LIN {X 0,Y 411.191,Z 465.266,A -85,B 0,C 180,E1 -10409.152,E2 -10409.152} C_VEL
LIN {X 0,Y 411.26,Z 465.255,A -85,B 0,C 180,E1 -10412.522,E2 -10412.522} C_VEL
LIN {X 0,Y 411.229,Z 465.262,A -85,B 0,C 180,E1 -10415.784,E2 -10415.784} C_VEL
LIN {X 0,Y 411.198,Z 465.264,A -85,B 0,C 180,E1 -10418.966,E2 -10418.966} C_VEL
LIN {X 0,Y 411.254,Z 465.257,A -85,B 0,C 180,E1 -10422.085,E2 -10422.085} C_VEL
LIN {X 0,Y 411.262,Z 465.258,A -85,B 0,C 180,E1 -10425.147,E2 -10425.147} C_VEL
LIN {X 0,Y 411.285,Z 465.252,A -85,B 0,C 180,E1 -10428.167,E2 -10428.167} C_VEL
LIN {X 0,Y 411.483,Z 465.229,A -85,B 0,C 180,E1 -10432.146,E2 -10432.146} C_VEL
LIN {X 0,Y 411.476,Z 465.229,A -85,B 0,C 180,E1 -10434.118,E2 -10434.118} C_VEL
LIN {X 0,Y 411.515,Z 465.226,A -85,B 0,C 180,E1 -10438.042,E2 -10438.042} C_VEL
LIN {X 0,Y 411.643,Z 465.21,A -85,B 0,C 180,E1 -10440,E2 -10440} C_VEL
LIN {X 0,Y 411.459,Z 465.231,A -85,B 0,C 180,E1 -10442.937,E2 -10442.937} C_VEL
LIN {X 0,Y 411.461,Z 465.232,A -85,B 0,C 180,E1 -10446.867,E2 -10446.867} C_VEL
LIN {X 0,Y 411.293,Z 465.252,A -85,B 0,C 180,E1 -10449.839,E2 -10449.839} C_VEL
LIN {X 0,Y 411.306,Z 465.253,A -85,B 0,C 180,E1 -10453.104,E2 -10453.104} C_VEL
LIN {X 0,Y 411.263,Z 465.255,A -85,B 0,C 180,E1 -10456.869,E2 -10456.869} C_VEL
LIN {X 0,Y 411.231,Z 465.261,A -85,B 0,C 180,E1 -10459.987,E2 -10459.987} C_VEL
LIN {X 0,Y 411.204,Z 465.264,A -85,B 0,C 180,E1 -10463.147,E2 -10463.147} C_VEL
LIN {X 0,Y 411.238,Z 465.258,A -85,B 0,C 180,E1 -10466.381,E2 -10466.381} C_VEL
LIN {X 0,Y 411.2,Z 465.266,A -85,B 0,C 180,E1 -10469.713,E2 -10469.713} C_VEL
LIN {X 0,Y 411.206,Z 465.266,A -85,B 0,C 180,E1 -10473.156,E2 -10473.156} C_VEL
LIN {X 0,Y 411.195,Z 465.264,A -85,B 0,C 180,E1 -10476.553,E2 -10476.553} C_VEL
LIN {X 0,Y 411.217,Z 465.262,A -85,B 0,C 180,E1 -10479.729,E2 -10479.729} C_VEL
LIN {X 0,Y 411.231,Z 465.262,A -85,B 0,C 180,E1 -10483.126,E2 -10483.126} C_VEL
LIN {X 0,Y 411.172,Z 465.275,A -85,B 0,C 180,E1 -10485.881,E2 -10485.881} C_VEL
LIN {X 0,Y 411.284,Z 465.464,A -85,B 0,C 180,E1 -10487.44,E2 -10487.44} C_VEL
LIN {X 0,Y 412.469,Z 472.197,A -85,B 0,C 180,E1 -10490.918,E2 -10490.918} C_VEL
LIN {X 0,Y 413.284,Z 477.387,A -85,B 0,C 180,E1 -10493.474,E2 -10493.474} C_VEL
LIN {X 0,Y 413.079,Z 482.509,A -85,B 0,C 180,E1 -10495.844,E2 -10495.844} C_VEL
LIN {X 0,Y 412.407,Z 490.177,A -85,B 0,C 180,E1 -10499.254,E2 -10499.254} C_VEL
LIN {X 0,Y 411.822,Z 497.821,A -85,B 0,C 180,E1 -10502.563,E2 -10502.563} C_VEL
LIN {X 0,Y 411.283,Z 505.453,A -85,B 0,C 180,E1 -10505.788,E2 -10505.788} C_VEL
LIN {X 0,Y 410.808,Z 514.359,A -85,B 0,C 180,E1 -10509.47,E2 -10509.47} C_VEL
LIN {X 0,Y 410.523,Z 522.363,A -85,B 0,C 180,E1 -10512.726,E2 -10512.726} C_VEL
LIN {X 0,Y 412.529,Z 536.719,A -85,B 0,C 180,E1 -10513.296,E2 -10513.296} C_VEL
LIN {X 0,Y 413.816,Z 548.267,A -85,B 0,C 180,E1 -10513.913,E2 -10513.913} C_VEL
LIN {X 0,Y 414.068,Z 553.582,A -85,B 0,C 180,E1 -10514.243,E2 -10514.243} C_VEL
LIN {X 0,Y 413.319,Z 565.526,A -85,B 0,C 180,E1 -10515.097,E2 -10515.097} C_VEL
LIN {X 0,Y 412.57,Z 576.424,A -85,B 0,C 180,E1 -10516.077,E2 -10516.077} C_VEL
LIN {X 0,Y 411.928,Z 586.371,A -85,B 0,C 180,E1 -10517.186,E2 -10517.186} C_VEL
LIN {X 0,Y 411.336,Z 595.435,A -85,B 0,C 180,E1 -10518.419,E2 -10518.419} C_VEL
LIN {X 0,Y 410.758,Z 604.315,A -85,B 0,C 180,E1 -10519.9,E2 -10519.9} C_VEL
LIN {X 0,Y 410.401,Z 611.44,A -85,B 0,C 180,E1 -10521.382,E2 -10521.382} C_VEL
LIN {X 0,Y 410.162,Z 617.937,A -85,B 0,C 180,E1 -10523.111,E2 -10523.111} C_VEL
LIN {X 0,Y 410.08,Z 622.193,A -85,B 0,C 180,E1 -10524.591,E2 -10524.591} C_VEL
LIN {X 0,Y 409.976,Z 625.337,A -85,B 0,C 180,E1 -10526.068,E2 -10526.068} C_VEL
LIN {X 0,Y 410.07,Z 626.893,A -85,B 0,C 180,E1 -10527.053,E2 -10527.053} C_VEL
LIN {X 0,Y 410.058,Z 627.975,A -85,B 0,C 180,E1 -10528.036,E2 -10528.036} C_VEL
LIN {X 0,Y 410.037,Z 628.624,A -85,B 0,C 180,E1 -10529.018,E2 -10529.018} C_VEL
LIN {X 0,Y 410.047,Z 628.868,A -85,B 0,C 180,E1 -10530,E2 -10530} C_VEL
LIN {X 0,Y 410.026,Z 628.7,A -85,B 0,C 180,E1 -10530.982,E2 -10530.982} C_VEL
LIN {X 0,Y 410.059,Z 628.077,A -85,B 0,C 180,E1 -10531.965,E2 -10531.965} C_VEL
LIN {X 0,Y 410.045,Z 627.032,A -85,B 0,C 180,E1 -10532.948,E2 -10532.948} C_VEL
LIN {X 0,Y 409.979,Z 625.569,A -85,B 0,C 180,E1 -10533.932,E2 -10533.932} C_VEL
LIN {X 0,Y 410.043,Z 622.528,A -85,B 0,C 180,E1 -10535.409,E2 -10535.409} C_VEL
LIN {X 0,Y 410.164,Z 618.421,A -85,B 0,C 180,E1 -10536.889,E2 -10536.889} C_VEL
LIN {X 0,Y 410.444,Z 612.154,A -85,B 0,C 180,E1 -10538.617,E2 -10538.617} C_VEL
LIN {X 0,Y 410.83,Z 604.043,A -85,B 0,C 180,E1 -10540.348,E2 -10540.348} C_VEL
LIN {X 0,Y 411.507,Z 595.34,A -85,B 0,C 180,E1 -10541.826,E2 -10541.826} C_VEL
LIN {X 0,Y 412.242,Z 584.879,A -85,B 0,C 180,E1 -10543.262,E2 -10543.262} C_VEL
LIN {X 0,Y 413.051,Z 574.993,A -85,B 0,C 180,E1 -10544.372,E2 -10544.372} C_VEL
LIN {X 0,Y 413.928,Z 563.907,A -85,B 0,C 180,E1 -10545.385,E2 -10545.385} C_VEL
LIN {X 0,Y 414.759,Z 552.383,A -85,B 0,C 180,E1 -10546.236,E2 -10546.236} C_VEL
LIN {X 0,Y 413.894,Z 539.48,A -85,B 0,C 180,E1 -10547.068,E2 -10547.068} C_VEL
LIN {X 0,Y 412.163,Z 526.898,A -85,B 0,C 180,E1 -10547.744,E2 -10547.744} C_VEL
LIN {X 0,Y 410.508,Z 518.922,A -85,B 0,C 180,E1 -10548.142,E2 -10548.142} C_VEL
LIN {X 0,Y 410.885,Z 510.509,A -85,B 0,C 180,E1 -10551.577,E2 -10551.577} C_VEL
LIN {X 0,Y 411.362,Z 501.923,A -85,B 0,C 180,E1 -10555.285,E2 -10555.285} C_VEL
LIN {X 0,Y 411.912,Z 494.917,A -85,B 0,C 180,E1 -10558.538,E2 -10558.538} C_VEL
LIN {X 0,Y 412.708,Z 488.374,A -85,B 0,C 180,E1 -10561.864,E2 -10561.864} C_VEL
LIN {X 0,Y 413.241,Z 484.363,A -85,B 0,C 180,E1 -10564.141,E2 -10564.141} C_VEL
LIN {X 0,Y 413.602,Z 480.707,A -85,B 0,C 180,E1 -10566.493,E2 -10566.493} C_VEL
LIN {X 0,Y 413.341,Z 477.537,A -85,B 0,C 180,E1 -10568.985,E2 -10568.985} C_VEL
LIN {X 0,Y 412.897,Z 474.939,A -85,B 0,C 180,E1 -10571.593,E2 -10571.593} C_VEL
LIN {X 0,Y 412.566,Z 472.95,A -85,B 0,C 180,E1 -10574.319,E2 -10574.319} C_VEL
LIN {X 0,Y 412.337,Z 471.651,A -85,B 0,C 180,E1 -10577.131,E2 -10577.131} C_VEL
LIN {X 0,Y 412.148,Z 471.064,A -85,B 0,C 180,E1 -10580.117,E2 -10580.117} C_VEL
LIN {X 0,Y 412.09,Z 471.198,A -85,B 0,C 180,E1 -10583.351,E2 -10583.351} C_VEL
LIN {X 0,Y 411.907,Z 471.748,A -85,B 0,C 180,E1 -10585.733,E2 -10585.733} C_VEL
LIN {X 0,Y 411.595,Z 473.076,A -85,B 0,C 180,E1 -10589.186,E2 -10589.186} C_VEL
LIN {X 0,Y 411.225,Z 474.94,A -85,B 0,C 180,E1 -10592.711,E2 -10592.711} C_VEL
LIN {X 0,Y 411.017,Z 476.852,A -85,B 0,C 180,E1 -10595.772,E2 -10595.772} C_VEL
LIN {X 0,Y 410.796,Z 479.083,A -85,B 0,C 180,E1 -10598.945,E2 -10598.945} C_VEL
LIN {X 0,Y 410.677,Z 481.366,A -85,B 0,C 180,E1 -10601.93,E2 -10601.93} C_VEL
LIN {X 0,Y 410.687,Z 481.441,A -85,B 0,C 180,E1 -10602.027,E2 -10602.027} C_VEL
LIN {X 0,Y 414.674,Z 493.731,A -85,B 0,C 180,E1 -10602.821,E2 -10602.821} C_VEL
LIN {X 0,Y 416.29,Z 500.968,A -85,B 0,C 180,E1 -10603.322,E2 -10603.322} C_VEL
LIN {X 0,Y 415.591,Z 513.919,A -85,B 0,C 180,E1 -10604.176,E2 -10604.176} C_VEL
LIN {X 0,Y 414.731,Z 524.949,A -85,B 0,C 180,E1 -10605.093,E2 -10605.093} C_VEL
LIN {X 0,Y 413.829,Z 536.039,A -85,B 0,C 180,E1 -10606.246,E2 -10606.246} C_VEL
LIN {X 0,Y 413.001,Z 545.517,A -85,B 0,C 180,E1 -10607.469,E2 -10607.469} C_VEL
LIN {X 0,Y 412.185,Z 554.785,A -85,B 0,C 180,E1 -10608.941,E2 -10608.941} C_VEL
LIN {X 0,Y 411.616,Z 562.199,A -85,B 0,C 180,E1 -10610.417,E2 -10610.417} C_VEL
LIN {X 0,Y 410.989,Z 569.077,A -85,B 0,C 180,E1 -10612.137,E2 -10612.137} C_VEL
LIN {X 0,Y 410.654,Z 573.62,A -85,B 0,C 180,E1 -10613.613,E2 -10613.613} C_VEL
LIN {X 0,Y 410.457,Z 577.055,A -85,B 0,C 180,E1 -10615.089,E2 -10615.089} C_VEL
LIN {X 0,Y 410.368,Z 578.784,A -85,B 0,C 180,E1 -10616.072,E2 -10616.072} C_VEL
LIN {X 0,Y 410.177,Z 580.949,A -85,B 0,C 180,E1 -10618.036,E2 -10618.036} C_VEL
LIN {X 0,Y 410.099,Z 581.44,A -85,B 0,C 180,E1 -10619.018,E2 -10619.018} C_VEL
LIN {X 0,Y 410.049,Z 581.491,A -85,B 0,C 180,E1 -10620,E2 -10620} C_VEL
LIN {X 0,Y 410.105,Z 580.377,A -85,B 0,C 180,E1 -10621.964,E2 -10621.964} C_VEL
LIN {X 0,Y 410.204,Z 579.217,A -85,B 0,C 180,E1 -10622.946,E2 -10622.946} C_VEL
LIN {X 0,Y 410.218,Z 576.654,A -85,B 0,C 180,E1 -10624.422,E2 -10624.422} C_VEL
LIN {X 0,Y 410.415,Z 573.064,A -85,B 0,C 180,E1 -10625.898,E2 -10625.898} C_VEL
LIN {X 0,Y 410.674,Z 568.359,A -85,B 0,C 180,E1 -10627.374,E2 -10627.374} C_VEL
LIN {X 0,Y 411.044,Z 561.242,A -85,B 0,C 180,E1 -10629.1,E2 -10629.1} C_VEL
LIN {X 0,Y 411.535,Z 553.565,A -85,B 0,C 180,E1 -10630.579,E2 -10630.579} C_VEL
LIN {X 0,Y 412.05,Z 545.74,A -85,B 0,C 180,E1 -10631.811,E2 -10631.811} C_VEL
LIN {X 0,Y 412.867,Z 535.163,A -85,B 0,C 180,E1 -10633.161,E2 -10633.161} C_VEL
LIN {X 0,Y 413.488,Z 523.691,A -85,B 0,C 180,E1 -10634.343,E2 -10634.343} C_VEL
LIN {X 0,Y 414.1,Z 512.559,A -85,B 0,C 180,E1 -10635.252,E2 -10635.252} C_VEL
LIN {X 0,Y 414.79,Z 499.262,A -85,B 0,C 180,E1 -10636.098,E2 -10636.098} C_VEL
LIN {X 0,Y 412.292,Z 486.848,A -85,B 0,C 180,E1 -10636.781,E2 -10636.781} C_VEL
LIN {X 0,Y 410.179,Z 477.539,A -85,B 0,C 180,E1 -10637.199,E2 -10637.199} C_VEL
LIN {X 0,Y 410.212,Z 474.54,A -85,B 0,C 180,E1 -10640.039,E2 -10640.039} C_VEL
LIN {X 0,Y 410.261,Z 471.258,A -85,B 0,C 180,E1 -10643.204,E2 -10643.204} C_VEL
LIN {X 0,Y 410.376,Z 467.977,A -85,B 0,C 180,E1 -10646.441,E2 -10646.441} C_VEL
LIN {X 0,Y 410.439,Z 465.362,A -85,B 0,C 180,E1 -10649.157,E2 -10649.157} C_VEL
LIN {X 0,Y 410.748,Z 465.323,A -85,B 0,C 180,E1 -10652.034,E2 -10652.034} C_VEL
LIN {X 0,Y 411.08,Z 465.28,A -85,B 0,C 180,E1 -10654.852,E2 -10654.852} C_VEL
LIN {X 0,Y 411.206,Z 465.265,A -85,B 0,C 180,E1 -10658.168,E2 -10658.168} C_VEL
LIN {X 0,Y 411.168,Z 465.267,A -85,B 0,C 180,E1 -10661.228,E2 -10661.228} C_VEL
LIN {X 0,Y 411.18,Z 465.269,A -85,B 0,C 180,E1 -10664.491,E2 -10664.491} C_VEL
LIN {X 0,Y 411.182,Z 465.268,A -85,B 0,C 180,E1 -10668.195,E2 -10668.195} C_VEL
LIN {X 0,Y 411.226,Z 465.261,A -85,B 0,C 180,E1 -10670.776,E2 -10670.776} C_VEL
LIN {X 0,Y 411.203,Z 465.264,A -85,B 0,C 180,E1 -10674.471,E2 -10674.471} C_VEL
LIN {X 0,Y 411.212,Z 465.263,A -85,B 0,C 180,E1 -10676.873,E2 -10676.873} C_VEL
LIN {X 0,Y 411.238,Z 465.259,A -85,B 0,C 180,E1 -10680.644,E2 -10680.644} C_VEL
LIN {X 0,Y 411.243,Z 465.26,A -85,B 0,C 180,E1 -10683.619,E2 -10683.619} C_VEL
LIN {X 0,Y 411.209,Z 465.261,A -85,B 0,C 180,E1 -10686.853,E2 -10686.853} C_VEL
LIN {X 0,Y 411.221,Z 465.263,A -85,B 0,C 180,E1 -10690.05,E2 -10690.05} C_VEL
LIN {X 0,Y 411.268,Z 465.254,A -85,B 0,C 180,E1 -10693.131,E2 -10693.131} C_VEL
LIN {X 0,Y 411.311,Z 465.249,A -85,B 0,C 180,E1 -10696.896,E2 -10696.896} C_VEL
LIN {X 0,Y 411.297,Z 465.255,A -85,B 0,C 180,E1 -10700.161,E2 -10700.161} C_VEL
LIN {X 0,Y 411.444,Z 465.232,A -85,B 0,C 180,E1 -10703.133,E2 -10703.133} C_VEL
LIN {X 0,Y 411.315,Z 465.249,A -85,B 0,C 180,E1 -10705.099,E2 -10705.099} C_VEL
LIN {X 0,Y 411.517,Z 465.227,A -85,B 0,C 180,E1 -10708.042,E2 -10708.042} C_VEL
LIN {X 0,Y 411.646,Z 465.211,A -85,B 0,C 180,E1 -10710,E2 -10710} C_VEL
LIN {X 0,Y 411.462,Z 465.231,A -85,B 0,C 180,E1 -10712.937,E2 -10712.937} C_VEL
LIN {X 0,Y 411.464,Z 465.233,A -85,B 0,C 180,E1 -10715.882,E2 -10715.882} C_VEL
LIN {X 0,Y 411.357,Z 465.244,A -85,B 0,C 180,E1 -10718.845,E2 -10718.845} C_VEL
LIN {X 0,Y 411.29,Z 465.254,A -85,B 0,C 180,E1 -10721.832,E2 -10721.832} C_VEL
LIN {X 0,Y 411.27,Z 465.256,A -85,B 0,C 180,E1 -10723.585,E2 -10723.585} C_VEL
LIN {X 0,Y 410.573,Z 465.346,A -85,B 0,C 180,E1 -10724.403,E2 -10724.403} C_VEL
LIN {X 0,Y 407.695,Z 465.703,A -85,B 0,C 180,E1 -10725.731,E2 -10725.731} C_VEL
LIN {X 0,Y 405.286,Z 466,A -85,B 0,C 180,E1 -10726.804,E2 -10726.804} C_VEL
LIN {X 0,Y 404.272,Z 466.129,A -85,B 0,C 180,E1 -10727.633,E2 -10727.633} C_VEL
LIN {X 0,Y 404.198,Z 466.136,A -85,B 0,C 180,E1 -10727.914,E2 -10727.914} C_VEL
LIN {X 0,Y 404.168,Z 466.139,A -85,B 0,C 180,E1 -10730.351,E2 -10730.351} C_VEL
LIN {X 0,Y 404.174,Z 466.142,A -85,B 0,C 180,E1 -10733.574,E2 -10733.574} C_VEL
LIN {X 0,Y 404.188,Z 466.139,A -85,B 0,C 180,E1 -10735.766,E2 -10735.766} C_VEL
LIN {X 0,Y 404.199,Z 466.138,A -85,B 0,C 180,E1 -10737.999,E2 -10737.999} C_VEL
LIN {X 0,Y 404.143,Z 466.145,A -85,B 0,C 180,E1 -10741.558,E2 -10741.558} C_VEL
LIN {X 0,Y 404.189,Z 466.135,A -85,B 0,C 180,E1 -10745.016,E2 -10745.016} C_VEL
LIN {X 0,Y 404.161,Z 466.14,A -85,B 0,C 180,E1 -10748.756,E2 -10748.756} C_VEL
LIN {X 0,Y 404.126,Z 466.147,A -85,B 0,C 180,E1 -10751.599,E2 -10751.599} C_VEL
LIN {X 0,Y 404.15,Z 466.142,A -85,B 0,C 180,E1 -10754.522,E2 -10754.522} C_VEL
LIN {X 0,Y 404.142,Z 466.144,A -85,B 0,C 180,E1 -10757.296,E2 -10757.296} C_VEL
LIN {X 0,Y 404.171,Z 466.141,A -85,B 0,C 180,E1 -10759.955,E2 -10759.955} C_VEL
LIN {X 0,Y 404.141,Z 466.144,A -85,B 0,C 180,E1 -10763.124,E2 -10763.124} C_VEL
LIN {X 0,Y 404.147,Z 466.142,A -85,B 0,C 180,E1 -10766.187,E2 -10766.187} C_VEL
LIN {X 0,Y 404.147,Z 466.144,A -85,B 0,C 180,E1 -10769.715,E2 -10769.715} C_VEL
LIN {X 0,Y 404.197,Z 466.136,A -85,B 0,C 180,E1 -10773.123,E2 -10773.123} C_VEL
LIN {X 0,Y 404.179,Z 466.14,A -85,B 0,C 180,E1 -10775.334,E2 -10775.334} C_VEL
LIN {X 0,Y 404.14,Z 466.142,A -85,B 0,C 180,E1 -10778.58,E2 -10778.58} C_VEL
LIN {X 0,Y 404.212,Z 466.136,A -85,B 0,C 180,E1 -10781.762,E2 -10781.762} C_VEL
LIN {X 0,Y 404.208,Z 466.135,A -85,B 0,C 180,E1 -10784.882,E2 -10784.882} C_VEL
LIN {X 0,Y 404.258,Z 466.129,A -85,B 0,C 180,E1 -10787.958,E2 -10787.958} C_VEL
LIN {X 0,Y 404.434,Z 466.107,A -85,B 0,C 180,E1 -10792.099,E2 -10792.099} C_VEL
LIN {X 0,Y 404.425,Z 466.108,A -85,B 0,C 180,E1 -10794.015,E2 -10794.015} C_VEL
LIN {X 0,Y 404.484,Z 466.102,A -85,B 0,C 180,E1 -10798.008,E2 -10798.008} C_VEL
LIN {X 0,Y 404.613,Z 466.085,A -85,B 0,C 180,E1 -10800,E2 -10800} C_VEL
LIN {X 0,Y 404.417,Z 466.108,A -85,B 0,C 180,E1 -10802.988,E2 -10802.988} C_VEL
LIN {X 0,Y 404.413,Z 466.111,A -85,B 0,C 180,E1 -10806.987,E2 -10806.987} C_VEL
LIN {X 0,Y 404.259,Z 466.127,A -85,B 0,C 180,E1 -10810.012,E2 -10810.012} C_VEL
LIN {X 0,Y 404.266,Z 466.13,A -85,B 0,C 180,E1 -10813.211,E2 -10813.211} C_VEL
LIN {X 0,Y 404.216,Z 466.134,A -85,B 0,C 180,E1 -10817.007,E2 -10817.007} C_VEL
LIN {X 0,Y 404.164,Z 466.14,A -85,B 0,C 180,E1 -10820.351,E2 -10820.351} C_VEL
LIN {X 0,Y 404.17,Z 466.142,A -85,B 0,C 180,E1 -10823.574,E2 -10823.574} C_VEL
LIN {X 0,Y 404.184,Z 466.138,A -85,B 0,C 180,E1 -10825.766,E2 -10825.766} C_VEL
LIN {X 0,Y 404.195,Z 466.137,A -85,B 0,C 180,E1 -10828,E2 -10828} C_VEL
LIN {X 0,Y 404.139,Z 466.145,A -85,B 0,C 180,E1 -10831.558,E2 -10831.558} C_VEL
LIN {X 0,Y 404.186,Z 466.14,A -85,B 0,C 180,E1 -10835.016,E2 -10835.016} C_VEL
LIN {X 0,Y 404.158,Z 466.14,A -85,B 0,C 180,E1 -10838.757,E2 -10838.757} C_VEL
LIN {X 0,Y 404.189,Z 466.139,A -85,B 0,C 180,E1 -10841.61,E2 -10841.61} C_VEL
LIN {X 0,Y 404.193,Z 466.141,A -85,B 0,C 180,E1 -10844.529,E2 -10844.529} C_VEL
LIN {X 0,Y 404.188,Z 466.205,A -85,B 0,C 180,E1 -10847.108,E2 -10847.108} C_VEL
LIN {X 0,Y 405.187,Z 471.8,A -85,B 0,C 180,E1 -10850.076,E2 -10850.076} C_VEL
LIN {X 0,Y 406.085,Z 477.086,A -85,B 0,C 180,E1 -10852.76,E2 -10852.76} C_VEL
LIN {X 0,Y 406.296,Z 480.457,A -85,B 0,C 180,E1 -10854.39,E2 -10854.39} C_VEL
LIN {X 0,Y 405.71,Z 487.242,A -85,B 0,C 180,E1 -10857.52,E2 -10857.52} C_VEL
LIN {X 0,Y 405.066,Z 494.883,A -85,B 0,C 180,E1 -10860.935,E2 -10860.935} C_VEL
LIN {X 0,Y 404.407,Z 503.418,A -85,B 0,C 180,E1 -10864.647,E2 -10864.647} C_VEL
LIN {X 0,Y 403.895,Z 511.378,A -85,B 0,C 180,E1 -10868.031,E2 -10868.031} C_VEL
LIN {X 0,Y 403.57,Z 518.976,A -85,B 0,C 180,E1 -10871.206,E2 -10871.206} C_VEL
LIN {X 0,Y 403.464,Z 522.056,A -85,B 0,C 180,E1 -10872.486,E2 -10872.486} C_VEL
LIN {X 0,Y 405.379,Z 536.008,A -85,B 0,C 180,E1 -10873.044,E2 -10873.044} C_VEL
LIN {X 0,Y 406.849,Z 549.029,A -85,B 0,C 180,E1 -10873.764,E2 -10873.764} C_VEL
LIN {X 0,Y 407.075,Z 554.128,A -85,B 0,C 180,E1 -10874.093,E2 -10874.093} C_VEL
LIN {X 0,Y 406.296,Z 565.865,A -85,B 0,C 180,E1 -10874.962,E2 -10874.962} C_VEL
LIN {X 0,Y 405.539,Z 576.607,A -85,B 0,C 180,E1 -10875.959,E2 -10875.959} C_VEL
LIN {X 0,Y 404.813,Z 587.399,A -85,B 0,C 180,E1 -10877.212,E2 -10877.212} C_VEL
LIN {X 0,Y 404.208,Z 596.23,A -85,B 0,C 180,E1 -10878.466,E2 -10878.466} C_VEL
LIN {X 0,Y 403.642,Z 604.871,A -85,B 0,C 180,E1 -10879.973,E2 -10879.973} C_VEL
LIN {X 0,Y 403.303,Z 611.789,A -85,B 0,C 180,E1 -10881.482,E2 -10881.482} C_VEL
LIN {X 0,Y 403.074,Z 617.317,A -85,B 0,C 180,E1 -10882.99,E2 -10882.99} C_VEL
LIN {X 0,Y 402.998,Z 621.624,A -85,B 0,C 180,E1 -10884.496,E2 -10884.496} C_VEL
LIN {X 0,Y 402.896,Z 624.813,A -85,B 0,C 180,E1 -10885.999,E2 -10885.999} C_VEL
LIN {X 0,Y 402.971,Z 626.388,A -85,B 0,C 180,E1 -10887.001,E2 -10887.001} C_VEL
LIN {X 0,Y 402.987,Z 627.509,A -85,B 0,C 180,E1 -10888.001,E2 -10888.001} C_VEL
LIN {X 0,Y 402.958,Z 628.174,A -85,B 0,C 180,E1 -10889.001,E2 -10889.001} C_VEL
LIN {X 0,Y 402.965,Z 628.432,A -85,B 0,C 180,E1 -10890,E2 -10890} C_VEL
LIN {X 0,Y 402.949,Z 628.281,A -85,B 0,C 180,E1 -10891,E2 -10891} C_VEL
LIN {X 0,Y 402.987,Z 627.687,A -85,B 0,C 180,E1 -10891.999,E2 -10891.999} C_VEL
LIN {X 0,Y 402.943,Z 626.654,A -85,B 0,C 180,E1 -10893,E2 -10893} C_VEL
LIN {X 0,Y 402.897,Z 625.206,A -85,B 0,C 180,E1 -10894.001,E2 -10894.001} C_VEL
LIN {X 0,Y 402.941,Z 622.189,A -85,B 0,C 180,E1 -10895.505,E2 -10895.505} C_VEL
LIN {X 0,Y 403.076,Z 618.118,A -85,B 0,C 180,E1 -10897.011,E2 -10897.011} C_VEL
LIN {X 0,Y 403.376,Z 611.914,A -85,B 0,C 180,E1 -10898.769,E2 -10898.769} C_VEL
LIN {X 0,Y 403.761,Z 605.127,A -85,B 0,C 180,E1 -10900.278,E2 -10900.278} C_VEL
LIN {X 0,Y 404.417,Z 596.794,A -85,B 0,C 180,E1 -10901.782,E2 -10901.782} C_VEL
LIN {X 0,Y 405.126,Z 586.865,A -85,B 0,C 180,E1 -10903.242,E2 -10903.242} C_VEL
LIN {X 0,Y 406.114,Z 575.952,A -85,B 0,C 180,E1 -10904.533,E2 -10904.533} C_VEL
LIN {X 0,Y 407.122,Z 564.319,A -85,B 0,C 180,E1 -10905.648,E2 -10905.648} C_VEL
LIN {X 0,Y 407.965,Z 553.078,A -85,B 0,C 180,E1 -10906.514,E2 -10906.514} C_VEL
LIN {X 0,Y 407.064,Z 538.698,A -85,B 0,C 180,E1 -10907.477,E2 -10907.477} C_VEL
LIN {X 0,Y 405.101,Z 526.011,A -85,B 0,C 180,E1 -10908.197,E2 -10908.197} C_VEL
LIN {X 0,Y 403.481,Z 518.343,A -85,B 0,C 180,E1 -10908.601,E2 -10908.601} C_VEL
LIN {X 0,Y 403.86,Z 510.337,A -85,B 0,C 180,E1 -10911.972,E2 -10911.972} C_VEL
LIN {X 0,Y 404.415,Z 501.848,A -85,B 0,C 180,E1 -10915.751,E2 -10915.751} C_VEL
LIN {X 0,Y 405.032,Z 494.957,A -85,B 0,C 180,E1 -10919.068,E2 -10919.068} C_VEL
LIN {X 0,Y 405.834,Z 488.572,A -85,B 0,C 180,E1 -10922.469,E2 -10922.469} C_VEL
LIN {X 0,Y 406.396,Z 484.677,A -85,B 0,C 180,E1 -10924.798,E2 -10924.798} C_VEL
LIN {X 0,Y 406.629,Z 481.021,A -85,B 0,C 180,E1 -10927.341,E2 -10927.341} C_VEL
LIN {X 0,Y 406.247,Z 478.175,A -85,B 0,C 180,E1 -10929.799,E2 -10929.799} C_VEL
LIN {X 0,Y 405.846,Z 475.767,A -85,B 0,C 180,E1 -10932.482,E2 -10932.482} C_VEL
LIN {X 0,Y 405.523,Z 473.983,A -85,B 0,C 180,E1 -10935.281,E2 -10935.281} C_VEL
LIN {X 0,Y 405.33,Z 472.878,A -85,B 0,C 180,E1 -10938.209,E2 -10938.209} C_VEL
LIN {X 0,Y 405.159,Z 472.502,A -85,B 0,C 180,E1 -10941.357,E2 -10941.357} C_VEL
LIN {X 0,Y 405.081,Z 472.695,A -85,B 0,C 180,E1 -10943.851,E2 -10943.851} C_VEL
LIN {X 0,Y 404.862,Z 473.312,A -85,B 0,C 180,E1 -10946.433,E2 -10946.433} C_VEL
LIN {X 0,Y 404.676,Z 474.1,A -85,B 0,C 180,E1 -10948.6,E2 -10948.6} C_VEL
LIN {X 0,Y 404.279,Z 475.734,A -85,B 0,C 180,E1 -10952.007,E2 -10952.007} C_VEL
LIN {X 0,Y 404.028,Z 477.682,A -85,B 0,C 180,E1 -10955.325,E2 -10955.325} C_VEL
LIN {X 0,Y 403.788,Z 479.852,A -85,B 0,C 180,E1 -10958.561,E2 -10958.561} C_VEL
LIN {X 0,Y 403.69,Z 482.098,A -85,B 0,C 180,E1 -10961.574,E2 -10961.574} C_VEL
LIN {X 0,Y 408.085,Z 495.368,A -85,B 0,C 180,E1 -10962.49,E2 -10962.49} C_VEL
LIN {X 0,Y 409.635,Z 501.868,A -85,B 0,C 180,E1 -10962.964,E2 -10962.964} C_VEL
LIN {X 0,Y 409.021,Z 513.996,A -85,B 0,C 180,E1 -10963.787,E2 -10963.787} C_VEL
LIN {X 0,Y 407.973,Z 526.749,A -85,B 0,C 180,E1 -10964.885,E2 -10964.885} C_VEL
LIN {X 0,Y 407.015,Z 537.107,A -85,B 0,C 180,E1 -10966.011,E2 -10966.011} C_VEL
LIN {X 0,Y 406.137,Z 546.494,A -85,B 0,C 180,E1 -10967.254,E2 -10967.254} C_VEL
LIN {X 0,Y 405.274,Z 555.668,A -85,B 0,C 180,E1 -10968.75,E2 -10968.75} C_VEL
LIN {X 0,Y 404.668,Z 562.987,A -85,B 0,C 180,E1 -10970.251,E2 -10970.251} C_VEL
LIN {X 0,Y 404.012,Z 569.765,A -85,B 0,C 180,E1 -10972.001,E2 -10972.001} C_VEL
LIN {X 0,Y 403.628,Z 574.24,A -85,B 0,C 180,E1 -10973.502,E2 -10973.502} C_VEL
LIN {X 0,Y 403.408,Z 577.636,A -85,B 0,C 180,E1 -10975.003,E2 -10975.003} C_VEL
LIN {X 0,Y 403.321,Z 579.322,A -85,B 0,C 180,E1 -10976.003,E2 -10976.003} C_VEL
LIN {X 0,Y 403.171,Z 580.584,A -85,B 0,C 180,E1 -10977.003,E2 -10977.003} C_VEL
LIN {X 0,Y 403.102,Z 581.443,A -85,B 0,C 180,E1 -10978.002,E2 -10978.002} C_VEL
LIN {X 0,Y 403.019,Z 581.901,A -85,B 0,C 180,E1 -10979.001,E2 -10979.001} C_VEL
LIN {X 0,Y 402.967,Z 581.914,A -85,B 0,C 180,E1 -10980,E2 -10980} C_VEL
LIN {X 0,Y 402.965,Z 581.528,A -85,B 0,C 180,E1 -10981,E2 -10981} C_VEL
LIN {X 0,Y 403.035,Z 580.743,A -85,B 0,C 180,E1 -10981.999,E2 -10981.999} C_VEL
LIN {X 0,Y 403.14,Z 579.537,A -85,B 0,C 180,E1 -10982.998,E2 -10982.998} C_VEL
LIN {X 0,Y 403.137,Z 576.926,A -85,B 0,C 180,E1 -10984.5,E2 -10984.5} C_VEL
LIN {X 0,Y 403.358,Z 573.28,A -85,B 0,C 180,E1 -10986.001,E2 -10986.001} C_VEL
LIN {X 0,Y 403.619,Z 568.506,A -85,B 0,C 180,E1 -10987.504,E2 -10987.504} C_VEL
LIN {X 0,Y 404.034,Z 561.323,A -85,B 0,C 180,E1 -10989.259,E2 -10989.259} C_VEL
LIN {X 0,Y 404.542,Z 553.568,A -85,B 0,C 180,E1 -10990.764,E2 -10990.764} C_VEL
LIN {X 0,Y 405.204,Z 543.857,A -85,B 0,C 180,E1 -10992.267,E2 -10992.267} C_VEL
LIN {X 0,Y 405.999,Z 533.913,A -85,B 0,C 180,E1 -10993.515,E2 -10993.515} C_VEL
LIN {X 0,Y 406.596,Z 523.244,A -85,B 0,C 180,E1 -10994.601,E2 -10994.601} C_VEL
LIN {X 0,Y 407.348,Z 510.399,A -85,B 0,C 180,E1 -10995.64,E2 -10995.64} C_VEL
LIN {X 0,Y 407.794,Z 499.436,A -85,B 0,C 180,E1 -10996.332,E2 -10996.332} C_VEL
LIN {X 0,Y 405.12,Z 487.017,A -85,B 0,C 180,E1 -10997.028,E2 -10997.028} C_VEL
LIN {X 0,Y 403.133,Z 477.889,A -85,B 0,C 180,E1 -10997.436,E2 -10997.436} C_VEL
LIN {X 0,Y 403.153,Z 474.777,A -85,B 0,C 180,E1 -11000.405,E2 -11000.405} C_VEL
LIN {X 0,Y 403.183,Z 471.466,A -85,B 0,C 180,E1 -11003.636,E2 -11003.636} C_VEL
LIN {X 0,Y 403.339,Z 468.144,A -85,B 0,C 180,E1 -11006.939,E2 -11006.939} C_VEL
LIN {X 0,Y 403.405,Z 466.238,A -85,B 0,C 180,E1 -11009.197,E2 -11009.197} C_VEL
LIN {X 0,Y 403.772,Z 466.192,A -85,B 0,C 180,E1 -11012.656,E2 -11012.656} C_VEL
LIN {X 0,Y 404.045,Z 466.155,A -85,B 0,C 180,E1 -11015.162,E2 -11015.162} C_VEL
LIN {X 0,Y 404.156,Z 466.143,A -85,B 0,C 180,E1 -11018.508,E2 -11018.508} C_VEL
LIN {X 0,Y 404.127,Z 466.145,A -85,B 0,C 180,E1 -11021.6,E2 -11021.6} C_VEL
LIN {X 0,Y 404.15,Z 466.144,A -85,B 0,C 180,E1 -11024.522,E2 -11024.522} C_VEL
LIN {X 0,Y 404.141,Z 466.142,A -85,B 0,C 180,E1 -11027.296,E2 -11027.296} C_VEL
LIN {X 0,Y 404.173,Z 466.141,A -85,B 0,C 180,E1 -11029.956,E2 -11029.956} C_VEL
LIN {X 0,Y 404.143,Z 466.14,A -85,B 0,C 180,E1 -11033.125,E2 -11033.125} C_VEL
LIN {X 0,Y 404.15,Z 466.144,A -85,B 0,C 180,E1 -11036.188,E2 -11036.188} C_VEL
LIN {X 0,Y 404.151,Z 466.142,A -85,B 0,C 180,E1 -11039.715,E2 -11039.715} C_VEL
LIN {X 0,Y 404.2,Z 466.135,A -85,B 0,C 180,E1 -11043.123,E2 -11043.123} C_VEL
LIN {X 0,Y 404.183,Z 466.137,A -85,B 0,C 180,E1 -11045.334,E2 -11045.334} C_VEL
LIN {X 0,Y 404.144,Z 466.143,A -85,B 0,C 180,E1 -11048.581,E2 -11048.581} C_VEL
LIN {X 0,Y 404.216,Z 466.135,A -85,B 0,C 180,E1 -11051.762,E2 -11051.762} C_VEL
LIN {X 0,Y 404.212,Z 466.132,A -85,B 0,C 180,E1 -11054.882,E2 -11054.882} C_VEL
LIN {X 0,Y 404.262,Z 466.13,A -85,B 0,C 180,E1 -11057.958,E2 -11057.958} C_VEL
LIN {X 0,Y 404.409,Z 466.112,A -85,B 0,C 180,E1 -11062.13,E2 -11062.13} C_VEL
LIN {X 0,Y 404.422,Z 466.11,A -85,B 0,C 180,E1 -11064.015,E2 -11064.015} C_VEL
LIN {X 0,Y 404.486,Z 466.103,A -85,B 0,C 180,E1 -11068.008,E2 -11068.008} C_VEL
LIN {X 0,Y 404.615,Z 466.087,A -85,B 0,C 180,E1 -11070,E2 -11070} C_VEL
LIN {X 0,Y 404.42,Z 466.108,A -85,B 0,C 180,E1 -11072.988,E2 -11072.988} C_VEL
LIN {X 0,Y 404.411,Z 466.113,A -85,B 0,C 180,E1 -11075.985,E2 -11075.985} C_VEL
LIN {X 0,Y 404.295,Z 466.123,A -85,B 0,C 180,E1 -11079.001,E2 -11079.001} C_VEL
LIN {X 0,Y 404.262,Z 466.131,A -85,B 0,C 180,E1 -11082.041,E2 -11082.041} C_VEL
LIN {X 0,Y 404.211,Z 466.133,A -85,B 0,C 180,E1 -11085.118,E2 -11085.118} C_VEL
LIN {X 0,Y 404.198,Z 466.136,A -85,B 0,C 180,E1 -11087.914,E2 -11087.914} C_VEL
LIN {X 0,Y 403.547,Z 466.221,A -85,B 0,C 180,E1 -11088.746,E2 -11088.746} C_VEL
LIN {X 0,Y 400.666,Z 466.582,A -85,B 0,C 180,E1 -11090.097,E2 -11090.097} C_VEL
LIN {X 0,Y 398.217,Z 466.885,A -85,B 0,C 180,E1 -11091.189,E2 -11091.189} C_VEL
LIN {X 0,Y 397.17,Z 467.013,A -85,B 0,C 180,E1 -11092.034,E2 -11092.034} C_VEL
LIN {X 0,Y 397.089,Z 467.021,A -85,B 0,C 180,E1 -11092.32,E2 -11092.32} C_VEL
LIN {X 0,Y 397.157,Z 467.014,A -85,B 0,C 180,E1 -11095.512,E2 -11095.512} C_VEL
LIN {X 0,Y 397.125,Z 467.016,A -85,B 0,C 180,E1 -11098.543,E2 -11098.543} C_VEL
LIN {X 0,Y 397.082,Z 467.025,A -85,B 0,C 180,E1 -11102.071,E2 -11102.071} C_VEL
LIN {X 0,Y 397.123,Z 467.018,A -85,B 0,C 180,E1 -11105.503,E2 -11105.503} C_VEL
LIN {X 0,Y 397.136,Z 467.015,A -85,B 0,C 180,E1 -11108.861,E2 -11108.861} C_VEL
LIN {X 0,Y 397.072,Z 467.023,A -85,B 0,C 180,E1 -11112.267,E2 -11112.267} C_VEL
LIN {X 0,Y 397.092,Z 467.021,A -85,B 0,C 180,E1 -11115.068,E2 -11115.068} C_VEL
LIN {X 0,Y 397.071,Z 467.026,A -85,B 0,C 180,E1 -11118.02,E2 -11118.02} C_VEL
LIN {X 0,Y 397.13,Z 467.016,A -85,B 0,C 180,E1 -11121.138,E2 -11121.138} C_VEL
LIN {X 0,Y 397.122,Z 467.017,A -85,B 0,C 180,E1 -11124.496,E2 -11124.496} C_VEL
LIN {X 0,Y 397.08,Z 467.024,A -85,B 0,C 180,E1 -11127.928,E2 -11127.928} C_VEL
LIN {X 0,Y 397.124,Z 467.019,A -85,B 0,C 180,E1 -11131.456,E2 -11131.456} C_VEL
LIN {X 0,Y 397.154,Z 467.011,A -85,B 0,C 180,E1 -11134.487,E2 -11134.487} C_VEL
LIN {X 0,Y 397.111,Z 467.019,A -85,B 0,C 180,E1 -11137.085,E2 -11137.085} C_VEL
LIN {X 0,Y 397.15,Z 467.012,A -85,B 0,C 180,E1 -11140.353,E2 -11140.353} C_VEL
LIN {X 0,Y 397.168,Z 467.014,A -85,B 0,C 180,E1 -11143.553,E2 -11143.553} C_VEL
LIN {X 0,Y 397.229,Z 467.003,A -85,B 0,C 180,E1 -11146.702,E2 -11146.702} C_VEL
LIN {X 0,Y 397.219,Z 467.006,A -85,B 0,C 180,E1 -11149.809,E2 -11149.809} C_VEL
LIN {X 0,Y 397.365,Z 466.987,A -85,B 0,C 180,E1 -11152.888,E2 -11152.888} C_VEL
LIN {X 0,Y 397.255,Z 467,A -85,B 0,C 180,E1 -11154.925,E2 -11154.925} C_VEL
LIN {X 0,Y 397.453,Z 466.977,A -85,B 0,C 180,E1 -11157.973,E2 -11157.973} C_VEL
LIN {X 0,Y 397.582,Z 466.961,A -85,B 0,C 180,E1 -11160,E2 -11160} C_VEL
LIN {X 0,Y 397.376,Z 466.986,A -85,B 0,C 180,E1 -11163.041,E2 -11163.041} C_VEL
LIN {X 0,Y 397.365,Z 466.989,A -85,B 0,C 180,E1 -11167.112,E2 -11167.112} C_VEL
LIN {X 0,Y 397.218,Z 467.003,A -85,B 0,C 180,E1 -11170.191,E2 -11170.191} C_VEL
LIN {X 0,Y 397.227,Z 467.006,A -85,B 0,C 180,E1 -11173.321,E2 -11173.321} C_VEL
LIN {X 0,Y 397.182,Z 467.011,A -85,B 0,C 180,E1 -11177.155,E2 -11177.155} C_VEL
LIN {X 0,Y 397.103,Z 467.02,A -85,B 0,C 180,E1 -11180.73,E2 -11180.73} C_VEL
LIN {X 0,Y 397.133,Z 467.015,A -85,B 0,C 180,E1 -11184.018,E2 -11184.018} C_VEL
LIN {X 0,Y 397.194,Z 467.01,A -85,B 0,C 180,E1 -11187.39,E2 -11187.39} C_VEL
LIN {X 0,Y 397.079,Z 467.023,A -85,B 0,C 180,E1 -11190.882,E2 -11190.882} C_VEL
LIN {X 0,Y 397.126,Z 467.016,A -85,B 0,C 180,E1 -11194.493,E2 -11194.493} C_VEL
LIN {X 0,Y 397.106,Z 467.017,A -85,B 0,C 180,E1 -11198.275,E2 -11198.275} C_VEL
LIN {X 0,Y 397.155,Z 467.013,A -85,B 0,C 180,E1 -11201.993,E2 -11201.993} C_VEL
LIN {X 0,Y 397.112,Z 467.024,A -85,B 0,C 180,E1 -11205.065,E2 -11205.065} C_VEL
LIN {X 0,Y 397.155,Z 467.052,A -85,B 0,C 180,E1 -11206.839,E2 -11206.839} C_VEL
LIN {X 0,Y 398.183,Z 472.885,A -85,B 0,C 180,E1 -11209.993,E2 -11209.993} C_VEL
LIN {X 0,Y 399.214,Z 479.191,A -85,B 0,C 180,E1 -11213.234,E2 -11213.234} C_VEL
LIN {X 0,Y 399.182,Z 483.03,A -85,B 0,C 180,E1 -11215.097,E2 -11215.097} C_VEL
LIN {X 0,Y 398.419,Z 490.667,A -85,B 0,C 180,E1 -11218.643,E2 -11218.643} C_VEL
LIN {X 0,Y 397.813,Z 498.192,A -85,B 0,C 180,E1 -11222.047,E2 -11222.047} C_VEL
LIN {X 0,Y 397.217,Z 505.874,A -85,B 0,C 180,E1 -11225.431,E2 -11225.431} C_VEL
LIN {X 0,Y 396.683,Z 514.71,A -85,B 0,C 180,E1 -11229.247,E2 -11229.247} C_VEL
LIN {X 0,Y 396.386,Z 521.768,A -85,B 0,C 180,E1 -11232.241,E2 -11232.241} C_VEL
LIN {X 0,Y 398.182,Z 535.066,A -85,B 0,C 180,E1 -11232.78,E2 -11232.78} C_VEL
LIN {X 0,Y 399.646,Z 547.854,A -85,B 0,C 180,E1 -11233.489,E2 -11233.489} C_VEL
LIN {X 0,Y 400.084,Z 554.596,A -85,B 0,C 180,E1 -11233.939,E2 -11233.939} C_VEL
LIN {X 0,Y 399.289,Z 566.146,A -85,B 0,C 180,E1 -11234.822,E2 -11234.822} C_VEL
LIN {X 0,Y 398.489,Z 576.85,A -85,B 0,C 180,E1 -11235.85,E2 -11235.85} C_VEL
LIN {X 0,Y 397.846,Z 586.447,A -85,B 0,C 180,E1 -11236.984,E2 -11236.984} C_VEL
LIN {X 0,Y 397.21,Z 595.362,A -85,B 0,C 180,E1 -11238.26,E2 -11238.26} C_VEL
LIN {X 0,Y 396.586,Z 604.104,A -85,B 0,C 180,E1 -11239.793,E2 -11239.793} C_VEL
LIN {X 0,Y 396.233,Z 611.091,A -85,B 0,C 180,E1 -11241.329,E2 -11241.329} C_VEL
LIN {X 0,Y 396.002,Z 616.677,A -85,B 0,C 180,E1 -11242.864,E2 -11242.864} C_VEL
LIN {X 0,Y 395.9,Z 621.034,A -85,B 0,C 180,E1 -11244.397,E2 -11244.397} C_VEL
LIN {X 0,Y 395.819,Z 624.272,A -85,B 0,C 180,E1 -11245.928,E2 -11245.928} C_VEL
LIN {X 0,Y 395.875,Z 625.867,A -85,B 0,C 180,E1 -11246.947,E2 -11246.947} C_VEL
LIN {X 0,Y 395.917,Z 627.029,A -85,B 0,C 180,E1 -11247.966,E2 -11247.966} C_VEL
LIN {X 0,Y 395.883,Z 627.716,A -85,B 0,C 180,E1 -11248.983,E2 -11248.983} C_VEL
LIN {X 0,Y 395.886,Z 627.993,A -85,B 0,C 180,E1 -11250,E2 -11250} C_VEL
LIN {X 0,Y 395.874,Z 627.859,A -85,B 0,C 180,E1 -11251.017,E2 -11251.017} C_VEL
LIN {X 0,Y 395.915,Z 627.301,A -85,B 0,C 180,E1 -11252.035,E2 -11252.035} C_VEL
LIN {X 0,Y 395.843,Z 626.282,A -85,B 0,C 180,E1 -11253.053,E2 -11253.053} C_VEL
LIN {X 0,Y 395.817,Z 624.853,A -85,B 0,C 180,E1 -11254.073,E2 -11254.073} C_VEL
LIN {X 0,Y 395.84,Z 621.371,A -85,B 0,C 180,E1 -11255.825,E2 -11255.825} C_VEL
LIN {X 0,Y 396.061,Z 616.251,A -85,B 0,C 180,E1 -11257.648,E2 -11257.648} C_VEL
LIN {X 0,Y 396.429,Z 609.6,A -85,B 0,C 180,E1 -11259.439,E2 -11259.439} C_VEL
LIN {X 0,Y 396.905,Z 602.433,A -85,B 0,C 180,E1 -11260.973,E2 -11260.973} C_VEL
LIN {X 0,Y 397.679,Z 593.584,A -85,B 0,C 180,E1 -11262.503,E2 -11262.503} C_VEL
LIN {X 0,Y 398.529,Z 583.543,A -85,B 0,C 180,E1 -11263.92,E2 -11263.92} C_VEL
LIN {X 0,Y 399.583,Z 572.655,A -85,B 0,C 180,E1 -11265.167,E2 -11265.167} C_VEL
LIN {X 0,Y 400.776,Z 560.352,A -85,B 0,C 180,E1 -11266.295,E2 -11266.295} C_VEL
LIN {X 0,Y 401.119,Z 552.139,A -85,B 0,C 180,E1 -11266.935,E2 -11266.935} C_VEL
LIN {X 0,Y 400.194,Z 537.83,A -85,B 0,C 180,E1 -11267.923,E2 -11267.923} C_VEL
LIN {X 0,Y 398.258,Z 525.872,A -85,B 0,C 180,E1 -11268.639,E2 -11268.639} C_VEL
LIN {X 0,Y 396.447,Z 517.799,A -85,B 0,C 180,E1 -11269.078,E2 -11269.078} C_VEL
LIN {X 0,Y 396.829,Z 510.177,A -85,B 0,C 180,E1 -11272.382,E2 -11272.382} C_VEL
LIN {X 0,Y 397.481,Z 501.811,A -85,B 0,C 180,E1 -11276.234,E2 -11276.234} C_VEL
LIN {X 0,Y 398.108,Z 495.048,A -85,B 0,C 180,E1 -11279.624,E2 -11279.624} C_VEL
LIN {X 0,Y 398.781,Z 490.29,A -85,B 0,C 180,E1 -11282.227,E2 -11282.227} C_VEL
LIN {X 0,Y 399.297,Z 486.87,A -85,B 0,C 180,E1 -11284.28,E2 -11284.28} C_VEL
LIN {X 0,Y 399.638,Z 483.3,A -85,B 0,C 180,E1 -11286.721,E2 -11286.721} C_VEL
LIN {X 0,Y 399.605,Z 481.69,A -85,B 0,C 180,E1 -11287.993,E2 -11287.993} C_VEL
LIN {X 0,Y 399.169,Z 478.74,A -85,B 0,C 180,E1 -11290.792,E2 -11290.792} C_VEL
LIN {X 0,Y 398.781,Z 476.438,A -85,B 0,C 180,E1 -11293.733,E2 -11293.733} C_VEL
LIN {X 0,Y 398.496,Z 474.968,A -85,B 0,C 180,E1 -11296.542,E2 -11296.542} C_VEL
LIN {X 0,Y 398.317,Z 474.174,A -85,B 0,C 180,E1 -11299.35,E2 -11299.35} C_VEL
LIN {X 0,Y 398.188,Z 473.984,A -85,B 0,C 180,E1 -11302.585,E2 -11302.585} C_VEL
LIN {X 0,Y 397.972,Z 474.445,A -85,B 0,C 180,E1 -11305.59,E2 -11305.59} C_VEL
LIN {X 0,Y 397.754,Z 475.182,A -85,B 0,C 180,E1 -11308.009,E2 -11308.009} C_VEL
LIN {X 0,Y 397.324,Z 476.688,A -85,B 0,C 180,E1 -11311.472,E2 -11311.472} C_VEL
LIN {X 0,Y 397.073,Z 478.538,A -85,B 0,C 180,E1 -11314.863,E2 -11314.863} C_VEL
LIN {X 0,Y 396.792,Z 480.662,A -85,B 0,C 180,E1 -11318.164,E2 -11318.164} C_VEL
LIN {X 0,Y 396.695,Z 482.729,A -85,B 0,C 180,E1 -11321.086,E2 -11321.086} C_VEL
LIN {X 0,Y 401.52,Z 496.964,A -85,B 0,C 180,E1 -11322.13,E2 -11322.13} C_VEL
LIN {X 0,Y 403.124,Z 504.019,A -85,B 0,C 180,E1 -11322.68,E2 -11322.68} C_VEL
LIN {X 0,Y 402.208,Z 517.289,A -85,B 0,C 180,E1 -11323.635,E2 -11323.635} C_VEL
LIN {X 0,Y 401.276,Z 528.125,A -85,B 0,C 180,E1 -11324.619,E2 -11324.619} C_VEL
LIN {X 0,Y 400.166,Z 539.362,A -85,B 0,C 180,E1 -11325.896,E2 -11325.896} C_VEL
LIN {X 0,Y 399.317,Z 547.551,A -85,B 0,C 180,E1 -11327.033,E2 -11327.033} C_VEL
LIN {X 0,Y 398.365,Z 556.537,A -85,B 0,C 180,E1 -11328.552,E2 -11328.552} C_VEL
LIN {X 0,Y 397.726,Z 563.789,A -85,B 0,C 180,E1 -11330.079,E2 -11330.079} C_VEL
LIN {X 0,Y 397.042,Z 570.505,A -85,B 0,C 180,E1 -11331.859,E2 -11331.859} C_VEL
LIN {X 0,Y 396.667,Z 574.352,A -85,B 0,C 180,E1 -11333.174,E2 -11333.174} C_VEL
LIN {X 0,Y 396.363,Z 578.241,A -85,B 0,C 180,E1 -11334.914,E2 -11334.914} C_VEL
LIN {X 0,Y 396.276,Z 579.873,A -85,B 0,C 180,E1 -11335.932,E2 -11335.932} C_VEL
LIN {X 0,Y 396.029,Z 581.936,A -85,B 0,C 180,E1 -11337.966,E2 -11337.966} C_VEL
LIN {X 0,Y 395.941,Z 582.353,A -85,B 0,C 180,E1 -11338.983,E2 -11338.983} C_VEL
LIN {X 0,Y 395.889,Z 582.335,A -85,B 0,C 180,E1 -11340,E2 -11340} C_VEL
LIN {X 0,Y 395.967,Z 581.106,A -85,B 0,C 180,E1 -11342.035,E2 -11342.035} C_VEL
LIN {X 0,Y 396.059,Z 579.848,A -85,B 0,C 180,E1 -11343.052,E2 -11343.052} C_VEL
LIN {X 0,Y 396.062,Z 577.176,A -85,B 0,C 180,E1 -11344.58,E2 -11344.58} C_VEL
LIN {X 0,Y 396.302,Z 573.462,A -85,B 0,C 180,E1 -11346.108,E2 -11346.108} C_VEL
LIN {X 0,Y 396.549,Z 568.613,A -85,B 0,C 180,E1 -11347.639,E2 -11347.639} C_VEL
LIN {X 0,Y 397.027,Z 561.345,A -85,B 0,C 180,E1 -11349.424,E2 -11349.424} C_VEL
LIN {X 0,Y 397.561,Z 553.465,A -85,B 0,C 180,E1 -11350.955,E2 -11350.955} C_VEL
LIN {X 0,Y 398.254,Z 543.643,A -85,B 0,C 180,E1 -11352.485,E2 -11352.485} C_VEL
LIN {X 0,Y 399.052,Z 533.545,A -85,B 0,C 180,E1 -11353.755,E2 -11353.755} C_VEL
LIN {X 0,Y 399.704,Z 521.922,A -85,B 0,C 180,E1 -11354.931,E2 -11354.931} C_VEL
LIN {X 0,Y 400.444,Z 509.613,A -85,B 0,C 180,E1 -11355.916,E2 -11355.916} C_VEL
LIN {X 0,Y 400.859,Z 500.465,A -85,B 0,C 180,E1 -11356.5,E2 -11356.5} C_VEL
LIN {X 0,Y 398.077,Z 487.52,A -85,B 0,C 180,E1 -11357.249,E2 -11357.249} C_VEL
LIN {X 0,Y 396.039,Z 478.229,A -85,B 0,C 180,E1 -11357.692,E2 -11357.692} C_VEL
LIN {X 0,Y 396.061,Z 475.009,A -85,B 0,C 180,E1 -11360.787,E2 -11360.787} C_VEL
LIN {X 0,Y 396.118,Z 471.665,A -85,B 0,C 180,E1 -11364.084,E2 -11364.084} C_VEL
LIN {X 0,Y 396.226,Z 469.424,A -85,B 0,C 180,E1 -11366.324,E2 -11366.324} C_VEL
LIN {X 0,Y 396.291,Z 467.175,A -85,B 0,C 180,E1 -11368.609,E2 -11368.609} C_VEL
LIN {X 0,Y 396.655,Z 467.079,A -85,B 0,C 180,E1 -11372.11,E2 -11372.11} C_VEL
LIN {X 0,Y 397.008,Z 467.031,A -85,B 0,C 180,E1 -11375.48,E2 -11375.48} C_VEL
LIN {X 0,Y 397.133,Z 467.015,A -85,B 0,C 180,E1 -11378.861,E2 -11378.861} C_VEL
LIN {X 0,Y 397.073,Z 467.025,A -85,B 0,C 180,E1 -11382.267,E2 -11382.267} C_VEL
LIN {X 0,Y 397.091,Z 467.019,A -85,B 0,C 180,E1 -11385.069,E2 -11385.069} C_VEL
LIN {X 0,Y 397.071,Z 467.027,A -85,B 0,C 180,E1 -11388.021,E2 -11388.021} C_VEL
LIN {X 0,Y 397.137,Z 467.014,A -85,B 0,C 180,E1 -11391.138,E2 -11391.138} C_VEL
LIN {X 0,Y 397.124,Z 467.018,A -85,B 0,C 180,E1 -11394.497,E2 -11394.497} C_VEL
LIN {X 0,Y 397.083,Z 467.024,A -85,B 0,C 180,E1 -11397.929,E2 -11397.929} C_VEL
LIN {X 0,Y 397.127,Z 467.016,A -85,B 0,C 180,E1 -11401.456,E2 -11401.456} C_VEL
LIN {X 0,Y 397.158,Z 467.015,A -85,B 0,C 180,E1 -11404.487,E2 -11404.487} C_VEL
LIN {X 0,Y 397.115,Z 467.016,A -85,B 0,C 180,E1 -11407.086,E2 -11407.086} C_VEL
LIN {X 0,Y 397.154,Z 467.015,A -85,B 0,C 180,E1 -11410.353,E2 -11410.353} C_VEL
LIN {X 0,Y 397.172,Z 467.011,A -85,B 0,C 180,E1 -11413.553,E2 -11413.553} C_VEL
LIN {X 0,Y 397.234,Z 467.003,A -85,B 0,C 180,E1 -11416.703,E2 -11416.703} C_VEL
LIN {X 0,Y 397.222,Z 467.006,A -85,B 0,C 180,E1 -11419.809,E2 -11419.809} C_VEL
LIN {X 0,Y 397.345,Z 466.988,A -85,B 0,C 180,E1 -11422.888,E2 -11422.888} C_VEL
LIN {X 0,Y 397.258,Z 467,A -85,B 0,C 180,E1 -11424.925,E2 -11424.925} C_VEL
LIN {X 0,Y 397.455,Z 466.978,A -85,B 0,C 180,E1 -11427.973,E2 -11427.973} C_VEL
LIN {X 0,Y 397.585,Z 466.963,A -85,B 0,C 180,E1 -11430,E2 -11430} C_VEL
LIN {X 0,Y 397.38,Z 466.984,A -85,B 0,C 180,E1 -11433.041,E2 -11433.041} C_VEL
LIN {X 0,Y 397.361,Z 466.99,A -85,B 0,C 180,E1 -11436.091,E2 -11436.091} C_VEL
LIN {X 0,Y 397.257,Z 467,A -85,B 0,C 180,E1 -11439.162,E2 -11439.162} C_VEL
LIN {X 0,Y 397.225,Z 467.006,A -85,B 0,C 180,E1 -11442.258,E2 -11442.258} C_VEL
LIN {X 0,Y 397.184,Z 467.01,A -85,B 0,C 180,E1 -11445.392,E2 -11445.392} C_VEL
LIN {X 0,Y 397.167,Z 467.011,A -85,B 0,C 180,E1 -11448.573,E2 -11448.573} C_VEL
LIN {X 0,Y 397.101,Z 467.023,A -85,B 0,C 180,E1 -11451.818,E2 -11451.818} C_VEL
LIN {X 0,Y 397.089,Z 467.021,A -85,B 0,C 180,E1 -11452.32,E2 -11452.32} C_VEL
LIN {X 0,Y 396.446,Z 467.102,A -85,B 0,C 180,E1 -11453.166,E2 -11453.166} C_VEL
LIN {X 0,Y 393.648,Z 467.45,A -85,B 0,C 180,E1 -11454.543,E2 -11454.543} C_VEL
LIN {X 0,Y 391.258,Z 467.749,A -85,B 0,C 180,E1 -11455.655,E2 -11455.655} C_VEL
LIN {X 0,Y 390.211,Z 467.878,A -85,B 0,C 180,E1 -11456.514,E2 -11456.514} C_VEL
LIN {X 0,Y 390.115,Z 467.888,A -85,B 0,C 180,E1 -11456.805,E2 -11456.805} C_VEL
LIN {X 0,Y 390.043,Z 467.9,A -85,B 0,C 180,E1 -11460.299,E2 -11460.299} C_VEL
LIN {X 0,Y 390.071,Z 467.898,A -85,B 0,C 180,E1 -11464.024,E2 -11464.024} C_VEL
LIN {X 0,Y 390.049,Z 467.901,A -85,B 0,C 180,E1 -11467.551,E2 -11467.551} C_VEL
LIN {X 0,Y 390.059,Z 467.896,A -85,B 0,C 180,E1 -11470.821,E2 -11470.821} C_VEL
LIN {X 0,Y 390.058,Z 467.899,A -85,B 0,C 180,E1 -11473.886,E2 -11473.886} C_VEL
LIN {X 0,Y 390.062,Z 467.896,A -85,B 0,C 180,E1 -11476.79,E2 -11476.79} C_VEL
LIN {X 0,Y 390.058,Z 467.899,A -85,B 0,C 180,E1 -11479.56,E2 -11479.56} C_VEL
LIN {X 0,Y 390.046,Z 467.898,A -85,B 0,C 180,E1 -11482.449,E2 -11482.449} C_VEL
LIN {X 0,Y 390.086,Z 467.894,A -85,B 0,C 180,E1 -11486.046,E2 -11486.046} C_VEL
LIN {X 0,Y 390.048,Z 467.9,A -85,B 0,C 180,E1 -11489.869,E2 -11489.869} C_VEL
LIN {X 0,Y 390.115,Z 467.891,A -85,B 0,C 180,E1 -11493.231,E2 -11493.231} C_VEL
LIN {X 0,Y 390.108,Z 467.89,A -85,B 0,C 180,E1 -11496.75,E2 -11496.75} C_VEL
LIN {X 0,Y 390.105,Z 467.892,A -85,B 0,C 180,E1 -11499.983,E2 -11499.983} C_VEL
LIN {X 0,Y 390.139,Z 467.889,A -85,B 0,C 180,E1 -11503.248,E2 -11503.248} C_VEL
LIN {X 0,Y 390.195,Z 467.879,A -85,B 0,C 180,E1 -11506.561,E2 -11506.561} C_VEL
LIN {X 0,Y 390.206,Z 467.878,A -85,B 0,C 180,E1 -11510.671,E2 -11510.671} C_VEL
LIN {X 0,Y 390.319,Z 467.864,A -85,B 0,C 180,E1 -11512.759,E2 -11512.759} C_VEL
LIN {X 0,Y 390.227,Z 467.875,A -85,B 0,C 180,E1 -11514.833,E2 -11514.833} C_VEL
LIN {X 0,Y 390.421,Z 467.853,A -85,B 0,C 180,E1 -11517.937,E2 -11517.937} C_VEL
LIN {X 0,Y 390.551,Z 467.837,A -85,B 0,C 180,E1 -11520,E2 -11520} C_VEL
LIN {X 0,Y 390.311,Z 467.866,A -85,B 0,C 180,E1 -11523.096,E2 -11523.096} C_VEL
LIN {X 0,Y 390.331,Z 467.863,A -85,B 0,C 180,E1 -11526.202,E2 -11526.202} C_VEL
LIN {X 0,Y 390.315,Z 467.864,A -85,B 0,C 180,E1 -11528.282,E2 -11528.282} C_VEL
LIN {X 0,Y 390.171,Z 467.882,A -85,B 0,C 180,E1 -11532.483,E2 -11532.483} C_VEL
LIN {X 0,Y 390.14,Z 467.889,A -85,B 0,C 180,E1 -11535.677,E2 -11535.677} C_VEL
LIN {X 0,Y 390.106,Z 467.891,A -85,B 0,C 180,E1 -11538.922,E2 -11538.922} C_VEL
LIN {X 0,Y 390.04,Z 467.898,A -85,B 0,C 180,E1 -11542.234,E2 -11542.234} C_VEL
LIN {X 0,Y 390.119,Z 467.89,A -85,B 0,C 180,E1 -11545.743,E2 -11545.743} C_VEL
LIN {X 0,Y 390.059,Z 467.899,A -85,B 0,C 180,E1 -11549.109,E2 -11549.109} C_VEL
LIN {X 0,Y 390.043,Z 467.898,A -85,B 0,C 180,E1 -11552.721,E2 -11552.721} C_VEL
LIN {X 0,Y 390.057,Z 467.898,A -85,B 0,C 180,E1 -11555.826,E2 -11555.826} C_VEL
LIN {X 0,Y 390.072,Z 467.899,A -85,B 0,C 180,E1 -11559.219,E2 -11559.219} C_VEL
LIN {X 0,Y 390.121,Z 467.888,A -85,B 0,C 180,E1 -11562.387,E2 -11562.387} C_VEL
LIN {X 0,Y 390.064,Z 467.904,A -85,B 0,C 180,E1 -11565.357,E2 -11565.357} C_VEL
LIN {X 0,Y 390.136,Z 468.064,A -85,B 0,C 180,E1 -11566.669,E2 -11566.669} C_VEL
LIN {X 0,Y 391.097,Z 473.549,A -85,B 0,C 180,E1 -11569.691,E2 -11569.691} C_VEL
LIN {X 0,Y 392.167,Z 480.05,A -85,B 0,C 180,E1 -11573.106,E2 -11573.106} C_VEL
LIN {X 0,Y 392.164,Z 483.9,A -85,B 0,C 180,E1 -11575.007,E2 -11575.007} C_VEL
LIN {X 0,Y 391.391,Z 491.519,A -85,B 0,C 180,E1 -11578.618,E2 -11578.618} C_VEL
LIN {X 0,Y 390.749,Z 499.113,A -85,B 0,C 180,E1 -11582.119,E2 -11582.119} C_VEL
LIN {X 0,Y 390.144,Z 506.688,A -85,B 0,C 180,E1 -11585.524,E2 -11585.524} C_VEL
LIN {X 0,Y 389.57,Z 515.378,A -85,B 0,C 180,E1 -11589.362,E2 -11589.362} C_VEL
LIN {X 0,Y 389.333,Z 521.523,A -85,B 0,C 180,E1 -11591.993,E2 -11591.993} C_VEL
LIN {X 0,Y 391.079,Z 534.764,A -85,B 0,C 180,E1 -11592.542,E2 -11592.542} C_VEL
LIN {X 0,Y 392.505,Z 546.574,A -85,B 0,C 180,E1 -11593.207,E2 -11593.207} C_VEL
LIN {X 0,Y 393.097,Z 554.943,A -85,B 0,C 180,E1 -11593.779,E2 -11593.779} C_VEL
LIN {X 0,Y 392.28,Z 566.327,A -85,B 0,C 180,E1 -11594.677,E2 -11594.677} C_VEL
LIN {X 0,Y 391.364,Z 578.135,A -85,B 0,C 180,E1 -11595.864,E2 -11595.864} C_VEL
LIN {X 0,Y 390.721,Z 587.376,A -85,B 0,C 180,E1 -11597.007,E2 -11597.007} C_VEL
LIN {X 0,Y 390.081,Z 596.076,A -85,B 0,C 180,E1 -11598.306,E2 -11598.306} C_VEL
LIN {X 0,Y 389.473,Z 604.561,A -85,B 0,C 180,E1 -11599.867,E2 -11599.867} C_VEL
LIN {X 0,Y 389.134,Z 611.391,A -85,B 0,C 180,E1 -11601.431,E2 -11601.431} C_VEL
LIN {X 0,Y 388.906,Z 617.644,A -85,B 0,C 180,E1 -11603.255,E2 -11603.255} C_VEL
LIN {X 0,Y 388.837,Z 621.673,A -85,B 0,C 180,E1 -11604.815,E2 -11604.815} C_VEL
LIN {X 0,Y 388.747,Z 623.719,A -85,B 0,C 180,E1 -11605.853,E2 -11605.853} C_VEL
LIN {X 0,Y 388.78,Z 625.335,A -85,B 0,C 180,E1 -11606.891,E2 -11606.891} C_VEL
LIN {X 0,Y 388.847,Z 626.53,A -85,B 0,C 180,E1 -11607.929,E2 -11607.929} C_VEL
LIN {X 0,Y 388.81,Z 627.253,A -85,B 0,C 180,E1 -11608.965,E2 -11608.965} C_VEL
LIN {X 0,Y 388.81,Z 627.55,A -85,B 0,C 180,E1 -11610,E2 -11610} C_VEL
LIN {X 0,Y 388.801,Z 627.436,A -85,B 0,C 180,E1 -11611.036,E2 -11611.036} C_VEL
LIN {X 0,Y 388.845,Z 626.912,A -85,B 0,C 180,E1 -11612.072,E2 -11612.072} C_VEL
LIN {X 0,Y 388.743,Z 625.918,A -85,B 0,C 180,E1 -11613.109,E2 -11613.109} C_VEL
LIN {X 0,Y 388.739,Z 624.508,A -85,B 0,C 180,E1 -11614.147,E2 -11614.147} C_VEL
LIN {X 0,Y 388.741,Z 621.419,A -85,B 0,C 180,E1 -11615.776,E2 -11615.776} C_VEL
LIN {X 0,Y 388.932,Z 617.582,A -85,B 0,C 180,E1 -11617.267,E2 -11617.267} C_VEL
LIN {X 0,Y 389.218,Z 612.461,A -85,B 0,C 180,E1 -11618.829,E2 -11618.829} C_VEL
LIN {X 0,Y 389.638,Z 606.07,A -85,B 0,C 180,E1 -11620.392,E2 -11620.392} C_VEL
LIN {X 0,Y 390.34,Z 598.223,A -85,B 0,C 180,E1 -11621.95,E2 -11621.95} C_VEL
LIN {X 0,Y 391.122,Z 588.528,A -85,B 0,C 180,E1 -11623.509,E2 -11623.509} C_VEL
LIN {X 0,Y 392.292,Z 577.653,A -85,B 0,C 180,E1 -11624.924,E2 -11624.924} C_VEL
LIN {X 0,Y 393.515,Z 565.338,A -85,B 0,C 180,E1 -11626.204,E2 -11626.204} C_VEL
LIN {X 0,Y 394.472,Z 554.768,A -85,B 0,C 180,E1 -11627.096,E2 -11627.096} C_VEL
LIN {X 0,Y 393.842,Z 541.578,A -85,B 0,C 180,E1 -11628.085,E2 -11628.085} C_VEL
LIN {X 0,Y 392.106,Z 529.043,A -85,B 0,C 180,E1 -11628.907,E2 -11628.907} C_VEL
LIN {X 0,Y 389.451,Z 517.138,A -85,B 0,C 180,E1 -11629.64,E2 -11629.64} C_VEL
LIN {X 0,Y 389.818,Z 510.265,A -85,B 0,C 180,E1 -11632.714,E2 -11632.714} C_VEL
LIN {X 0,Y 390.359,Z 503.674,A -85,B 0,C 180,E1 -11635.816,E2 -11635.816} C_VEL
LIN {X 0,Y 391.097,Z 496.234,A -85,B 0,C 180,E1 -11639.616,E2 -11639.616} C_VEL
LIN {X 0,Y 391.871,Z 491.031,A -85,B 0,C 180,E1 -11642.55,E2 -11642.55} C_VEL
LIN {X 0,Y 392.449,Z 487.212,A -85,B 0,C 180,E1 -11644.964,E2 -11644.964} C_VEL
LIN {X 0,Y 392.68,Z 485.232,A -85,B 0,C 180,E1 -11646.352,E2 -11646.352} C_VEL
LIN {X 0,Y 392.543,Z 482.258,A -85,B 0,C 180,E1 -11648.803,E2 -11648.803} C_VEL
LIN {X 0,Y 392.126,Z 479.63,A -85,B 0,C 180,E1 -11651.54,E2 -11651.54} C_VEL
LIN {X 0,Y 391.772,Z 477.585,A -85,B 0,C 180,E1 -11654.397,E2 -11654.397} C_VEL
LIN {X 0,Y 391.51,Z 476.206,A -85,B 0,C 180,E1 -11657.392,E2 -11657.392} C_VEL
LIN {X 0,Y 391.302,Z 475.517,A -85,B 0,C 180,E1 -11660.562,E2 -11660.562} C_VEL
LIN {X 0,Y 391.176,Z 475.523,A -85,B 0,C 180,E1 -11663.638,E2 -11663.638} C_VEL
LIN {X 0,Y 390.978,Z 475.956,A -85,B 0,C 180,E1 -11666.135,E2 -11666.135} C_VEL
LIN {X 0,Y 390.563,Z 477.165,A -85,B 0,C 180,E1 -11669.745,E2 -11669.745} C_VEL
LIN {X 0,Y 390.159,Z 478.822,A -85,B 0,C 180,E1 -11673.235,E2 -11673.235} C_VEL
LIN {X 0,Y 389.91,Z 480.896,A -85,B 0,C 180,E1 -11676.819,E2 -11676.819} C_VEL
LIN {X 0,Y 389.7,Z 483.382,A -85,B 0,C 180,E1 -11680.549,E2 -11680.549} C_VEL
LIN {X 0,Y 394.387,Z 496.846,A -85,B 0,C 180,E1 -11681.609,E2 -11681.609} C_VEL
LIN {X 0,Y 396.401,Z 504.348,A -85,B 0,C 180,E1 -11682.227,E2 -11682.227} C_VEL
LIN {X 0,Y 396.539,Z 507.53,A -85,B 0,C 180,E1 -11682.465,E2 -11682.465} C_VEL
LIN {X 0,Y 395.57,Z 519.161,A -85,B 0,C 180,E1 -11683.352,E2 -11683.352} C_VEL
LIN {X 0,Y 394.438,Z 530.942,A -85,B 0,C 180,E1 -11684.498,E2 -11684.498} C_VEL
LIN {X 0,Y 393.275,Z 541.601,A -85,B 0,C 180,E1 -11685.776,E2 -11685.776} C_VEL
LIN {X 0,Y 392.489,Z 548.688,A -85,B 0,C 180,E1 -11686.803,E2 -11686.803} C_VEL
LIN {X 0,Y 391.496,Z 557.528,A -85,B 0,C 180,E1 -11688.349,E2 -11688.349} C_VEL
LIN {X 0,Y 390.789,Z 564.645,A -85,B 0,C 180,E1 -11689.901,E2 -11689.901} C_VEL
LIN {X 0,Y 390.055,Z 571.233,A -85,B 0,C 180,E1 -11691.712,E2 -11691.712} C_VEL
LIN {X 0,Y 389.637,Z 575.213,A -85,B 0,C 180,E1 -11693.115,E2 -11693.115} C_VEL
LIN {X 0,Y 389.321,Z 578.854,A -85,B 0,C 180,E1 -11694.822,E2 -11694.822} C_VEL
LIN {X 0,Y 389.233,Z 580.45,A -85,B 0,C 180,E1 -11695.858,E2 -11695.858} C_VEL
LIN {X 0,Y 389.06,Z 581.651,A -85,B 0,C 180,E1 -11696.894,E2 -11696.894} C_VEL
LIN {X 0,Y 388.96,Z 582.45,A -85,B 0,C 180,E1 -11697.929,E2 -11697.929} C_VEL
LIN {X 0,Y 388.866,Z 582.808,A -85,B 0,C 180,E1 -11698.965,E2 -11698.965} C_VEL
LIN {X 0,Y 388.812,Z 582.757,A -85,B 0,C 180,E1 -11700,E2 -11700} C_VEL
LIN {X 0,Y 388.817,Z 582.311,A -85,B 0,C 180,E1 -11701.036,E2 -11701.036} C_VEL
LIN {X 0,Y 388.901,Z 581.459,A -85,B 0,C 180,E1 -11702.072,E2 -11702.072} C_VEL
LIN {X 0,Y 388.979,Z 580.155,A -85,B 0,C 180,E1 -11703.107,E2 -11703.107} C_VEL
LIN {X 0,Y 388.993,Z 577.422,A -85,B 0,C 180,E1 -11704.664,E2 -11704.664} C_VEL
LIN {X 0,Y 389.281,Z 572.843,A -85,B 0,C 180,E1 -11706.498,E2 -11706.498} C_VEL
LIN {X 0,Y 389.595,Z 566.823,A -85,B 0,C 180,E1 -11708.298,E2 -11708.298} C_VEL
LIN {X 0,Y 390.104,Z 560.131,A -85,B 0,C 180,E1 -11709.855,E2 -11709.855} C_VEL
LIN {X 0,Y 390.664,Z 551.845,A -85,B 0,C 180,E1 -11711.414,E2 -11711.414} C_VEL
LIN {X 0,Y 391.295,Z 543.426,A -85,B 0,C 180,E1 -11712.711,E2 -11712.711} C_VEL
LIN {X 0,Y 392.117,Z 533.146,A -85,B 0,C 180,E1 -11714.003,E2 -11714.003} C_VEL
LIN {X 0,Y 392.797,Z 521.468,A -85,B 0,C 180,E1 -11715.191,E2 -11715.191} C_VEL
LIN {X 0,Y 393.463,Z 510.623,A -85,B 0,C 180,E1 -11716.073,E2 -11716.073} C_VEL
LIN {X 0,Y 393.827,Z 501.011,A -85,B 0,C 180,E1 -11716.706,E2 -11716.706} C_VEL
LIN {X 0,Y 391.066,Z 488.304,A -85,B 0,C 180,E1 -11717.466,E2 -11717.466} C_VEL
LIN {X 0,Y 388.964,Z 478.596,A -85,B 0,C 180,E1 -11717.923,E2 -11717.923} C_VEL
LIN {X 0,Y 389.004,Z 475.238,A -85,B 0,C 180,E1 -11721.182,E2 -11721.182} C_VEL
LIN {X 0,Y 389.07,Z 471.846,A -85,B 0,C 180,E1 -11724.549,E2 -11724.549} C_VEL
LIN {X 0,Y 389.213,Z 468.447,A -85,B 0,C 180,E1 -11728.001,E2 -11728.001} C_VEL
LIN {X 0,Y 389.39,Z 467.984,A -85,B 0,C 180,E1 -11729.963,E2 -11729.963} C_VEL
LIN {X 0,Y 389.667,Z 467.948,A -85,B 0,C 180,E1 -11732.758,E2 -11732.758} C_VEL
LIN {X 0,Y 389.973,Z 467.909,A -85,B 0,C 180,E1 -11735.808,E2 -11735.808} C_VEL
LIN {X 0,Y 390.073,Z 467.893,A -85,B 0,C 180,E1 -11739.218,E2 -11739.218} C_VEL
LIN {X 0,Y 390.047,Z 467.901,A -85,B 0,C 180,E1 -11742.374,E2 -11742.374} C_VEL
LIN {X 0,Y 390.048,Z 467.896,A -85,B 0,C 180,E1 -11745.355,E2 -11745.355} C_VEL
LIN {X 0,Y 390.036,Z 467.902,A -85,B 0,C 180,E1 -11748.187,E2 -11748.187} C_VEL
LIN {X 0,Y 390.096,Z 467.892,A -85,B 0,C 180,E1 -11750.908,E2 -11750.908} C_VEL
LIN {X 0,Y 390.09,Z 467.893,A -85,B 0,C 180,E1 -11754.793,E2 -11754.793} C_VEL
LIN {X 0,Y 390.037,Z 467.901,A -85,B 0,C 180,E1 -11757.875,E2 -11757.875} C_VEL
LIN {X 0,Y 390.063,Z 467.895,A -85,B 0,C 180,E1 -11760.891,E2 -11760.891} C_VEL
LIN {X 0,Y 390.125,Z 467.891,A -85,B 0,C 180,E1 -11764.257,E2 -11764.257} C_VEL
LIN {X 0,Y 390.046,Z 467.899,A -85,B 0,C 180,E1 -11767.766,E2 -11767.766} C_VEL
LIN {X 0,Y 390.111,Z 467.89,A -85,B 0,C 180,E1 -11771.078,E2 -11771.078} C_VEL
LIN {X 0,Y 390.145,Z 467.888,A -85,B 0,C 180,E1 -11774.323,E2 -11774.323} C_VEL
LIN {X 0,Y 390.176,Z 467.883,A -85,B 0,C 180,E1 -11777.517,E2 -11777.517} C_VEL
LIN {X 0,Y 390.203,Z 467.878,A -85,B 0,C 180,E1 -11780.671,E2 -11780.671} C_VEL
LIN {X 0,Y 390.325,Z 467.866,A -85,B 0,C 180,E1 -11783.798,E2 -11783.798} C_VEL
LIN {X 0,Y 390.423,Z 467.854,A -85,B 0,C 180,E1 -11787.937,E2 -11787.937} C_VEL
LIN {X 0,Y 390.554,Z 467.839,A -85,B 0,C 180,E1 -11790,E2 -11790} C_VEL
LIN {X 0,Y 390.314,Z 467.864,A -85,B 0,C 180,E1 -11793.096,E2 -11793.096} C_VEL
LIN {X 0,Y 390.313,Z 467.867,A -85,B 0,C 180,E1 -11796.202,E2 -11796.202} C_VEL
LIN {X 0,Y 390.209,Z 467.878,A -85,B 0,C 180,E1 -11799.328,E2 -11799.328} C_VEL
LIN {X 0,Y 390.176,Z 467.882,A -85,B 0,C 180,E1 -11802.483,E2 -11802.483} C_VEL
LIN {X 0,Y 390.144,Z 467.889,A -85,B 0,C 180,E1 -11805.676,E2 -11805.676} C_VEL
LIN {X 0,Y 390.11,Z 467.889,A -85,B 0,C 180,E1 -11808.922,E2 -11808.922} C_VEL
LIN {X 0,Y 390.045,Z 467.899,A -85,B 0,C 180,E1 -11812.322,E2 -11812.322} C_VEL
LIN {X 0,Y 390.123,Z 467.891,A -85,B 0,C 180,E1 -11815.743,E2 -11815.743} C_VEL
LIN {X 0,Y 390.115,Z 467.888,A -85,B 0,C 180,E1 -11816.805,E2 -11816.805} C_VEL
LIN {X 0,Y 389.41,Z 467.98,A -85,B 0,C 180,E1 -11817.666,E2 -11817.666} C_VEL
LIN {X 0,Y 386.516,Z 468.337,A -85,B 0,C 180,E1 -11819.066,E2 -11819.066} C_VEL
LIN {X 0,Y 384.09,Z 468.642,A -85,B 0,C 180,E1 -11820.198,E2 -11820.198} C_VEL
LIN {X 0,Y 383.056,Z 468.769,A -85,B 0,C 180,E1 -11821.074,E2 -11821.074} C_VEL
LIN {X 0,Y 382.976,Z 468.777,A -85,B 0,C 180,E1 -11821.37,E2 -11821.37} C_VEL
LIN {X 0,Y 383.021,Z 468.772,A -85,B 0,C 180,E1 -11824.667,E2 -11824.667} C_VEL
LIN {X 0,Y 383.004,Z 468.778,A -85,B 0,C 180,E1 -11827.904,E2 -11827.904} C_VEL
LIN {X 0,Y 382.987,Z 468.779,A -85,B 0,C 180,E1 -11831.347,E2 -11831.347} C_VEL
LIN {X 0,Y 383,Z 468.777,A -85,B 0,C 180,E1 -11834.303,E2 -11834.303} C_VEL
LIN {X 0,Y 383.012,Z 468.776,A -85,B 0,C 180,E1 -11837.24,E2 -11837.24} C_VEL
LIN {X 0,Y 383.016,Z 468.773,A -85,B 0,C 180,E1 -11840.413,E2 -11840.413} C_VEL
LIN {X 0,Y 383.028,Z 468.775,A -85,B 0,C 180,E1 -11844.044,E2 -11844.044} C_VEL
LIN {X 0,Y 382.988,Z 468.781,A -85,B 0,C 180,E1 -11847.577,E2 -11847.577} C_VEL
LIN {X 0,Y 382.993,Z 468.777,A -85,B 0,C 180,E1 -11850.3,E2 -11850.3} C_VEL
LIN {X 0,Y 383.058,Z 468.768,A -85,B 0,C 180,E1 -11852.698,E2 -11852.698} C_VEL
LIN {X 0,Y 383.035,Z 468.772,A -85,B 0,C 180,E1 -11856.192,E2 -11856.192} C_VEL
LIN {X 0,Y 383.057,Z 468.772,A -85,B 0,C 180,E1 -11859.598,E2 -11859.598} C_VEL
LIN {X 0,Y 383.106,Z 468.762,A -85,B 0,C 180,E1 -11862.931,E2 -11862.931} C_VEL
LIN {X 0,Y 383.126,Z 468.759,A -85,B 0,C 180,E1 -11866.463,E2 -11866.463} C_VEL
LIN {X 0,Y 383.153,Z 468.756,A -85,B 0,C 180,E1 -11870.498,E2 -11870.498} C_VEL
LIN {X 0,Y 383.274,Z 468.741,A -85,B 0,C 180,E1 -11872.625,E2 -11872.625} C_VEL
LIN {X 0,Y 383.2,Z 468.75,A -85,B 0,C 180,E1 -11874.738,E2 -11874.738} C_VEL
LIN {X 0,Y 383.389,Z 468.729,A -85,B 0,C 180,E1 -11877.899,E2 -11877.899} C_VEL
LIN {X 0,Y 383.521,Z 468.712,A -85,B 0,C 180,E1 -11880,E2 -11880} C_VEL
LIN {X 0,Y 383.247,Z 468.746,A -85,B 0,C 180,E1 -11883.153,E2 -11883.153} C_VEL
LIN {X 0,Y 383.288,Z 468.74,A -85,B 0,C 180,E1 -11886.316,E2 -11886.316} C_VEL
LIN {X 0,Y 383.26,Z 468.742,A -85,B 0,C 180,E1 -11888.435,E2 -11888.435} C_VEL
LIN {X 0,Y 383.098,Z 468.766,A -85,B 0,C 180,E1 -11891.642,E2 -11891.642} C_VEL
LIN {X 0,Y 383.11,Z 468.763,A -85,B 0,C 180,E1 -11894.882,E2 -11894.882} C_VEL
LIN {X 0,Y 383.063,Z 468.767,A -85,B 0,C 180,E1 -11898.173,E2 -11898.173} C_VEL
LIN {X 0,Y 382.993,Z 468.78,A -85,B 0,C 180,E1 -11901.531,E2 -11901.531} C_VEL
LIN {X 0,Y 383.052,Z 468.77,A -85,B 0,C 180,E1 -11904.96,E2 -11904.96} C_VEL
LIN {X 0,Y 383.029,Z 468.772,A -85,B 0,C 180,E1 -11908.27,E2 -11908.27} C_VEL
LIN {X 0,Y 383.009,Z 468.773,A -85,B 0,C 180,E1 -11912.15,E2 -11912.15} C_VEL
LIN {X 0,Y 383.018,Z 468.774,A -85,B 0,C 180,E1 -11914.668,E2 -11914.668} C_VEL
LIN {X 0,Y 383.001,Z 468.775,A -85,B 0,C 180,E1 -11917.904,E2 -11917.904} C_VEL
LIN {X 0,Y 383.045,Z 468.773,A -85,B 0,C 180,E1 -11921.339,E2 -11921.339} C_VEL
LIN {X 0,Y 383.037,Z 468.777,A -85,B 0,C 180,E1 -11924.31,E2 -11924.31} C_VEL
LIN {X 0,Y 383.064,Z 468.991,A -85,B 0,C 180,E1 -11926.45,E2 -11926.45} C_VEL
LIN {X 0,Y 384.049,Z 474.381,A -85,B 0,C 180,E1 -11929.486,E2 -11929.486} C_VEL
LIN {X 0,Y 385.125,Z 480.888,A -85,B 0,C 180,E1 -11932.972,E2 -11932.972} C_VEL
LIN {X 0,Y 385.106,Z 485.33,A -85,B 0,C 180,E1 -11935.208,E2 -11935.208} C_VEL
LIN {X 0,Y 384.349,Z 492.333,A -85,B 0,C 180,E1 -11938.592,E2 -11938.592} C_VEL
LIN {X 0,Y 383.675,Z 499.914,A -85,B 0,C 180,E1 -11942.154,E2 -11942.154} C_VEL
LIN {X 0,Y 383.035,Z 507.461,A -85,B 0,C 180,E1 -11945.617,E2 -11945.617} C_VEL
LIN {X 0,Y 382.461,Z 516.263,A -85,B 0,C 180,E1 -11949.58,E2 -11949.58} C_VEL
LIN {X 0,Y 382.246,Z 521.058,A -85,B 0,C 180,E1 -11951.717,E2 -11951.717} C_VEL
LIN {X 0,Y 384.075,Z 535.084,A -85,B 0,C 180,E1 -11952.338,E2 -11952.338} C_VEL
LIN {X 0,Y 385.597,Z 548.146,A -85,B 0,C 180,E1 -11953.113,E2 -11953.113} C_VEL
LIN {X 0,Y 386.088,Z 555.165,A -85,B 0,C 180,E1 -11953.612,E2 -11953.612} C_VEL
LIN {X 0,Y 385.271,Z 566.385,A -85,B 0,C 180,E1 -11954.527,E2 -11954.527} C_VEL
LIN {X 0,Y 384.306,Z 578.239,A -85,B 0,C 180,E1 -11955.752,E2 -11955.752} C_VEL
LIN {X 0,Y 383.592,Z 588.224,A -85,B 0,C 180,E1 -11957.03,E2 -11957.03} C_VEL
LIN {X 0,Y 382.959,Z 596.681,A -85,B 0,C 180,E1 -11958.354,E2 -11958.354} C_VEL
LIN {X 0,Y 382.374,Z 604.958,A -85,B 0,C 180,E1 -11959.944,E2 -11959.944} C_VEL
LIN {X 0,Y 382.022,Z 611.64,A -85,B 0,C 180,E1 -11961.537,E2 -11961.537} C_VEL
LIN {X 0,Y 381.834,Z 616.955,A -85,B 0,C 180,E1 -11963.129,E2 -11963.129} C_VEL
LIN {X 0,Y 381.751,Z 621.053,A -85,B 0,C 180,E1 -11964.719,E2 -11964.719} C_VEL
LIN {X 0,Y 381.679,Z 623.15,A -85,B 0,C 180,E1 -11965.776,E2 -11965.776} C_VEL
LIN {X 0,Y 381.688,Z 624.791,A -85,B 0,C 180,E1 -11966.834,E2 -11966.834} C_VEL
LIN {X 0,Y 381.779,Z 626.013,A -85,B 0,C 180,E1 -11967.89,E2 -11967.89} C_VEL
LIN {X 0,Y 381.739,Z 626.785,A -85,B 0,C 180,E1 -11968.945,E2 -11968.945} C_VEL
LIN {X 0,Y 381.736,Z 627.104,A -85,B 0,C 180,E1 -11970,E2 -11970} C_VEL
LIN {X 0,Y 381.731,Z 627.014,A -85,B 0,C 180,E1 -11971.055,E2 -11971.055} C_VEL
LIN {X 0,Y 381.756,Z 626.514,A -85,B 0,C 180,E1 -11972.11,E2 -11972.11} C_VEL
LIN {X 0,Y 381.646,Z 625.565,A -85,B 0,C 180,E1 -11973.167,E2 -11973.167} C_VEL
LIN {X 0,Y 381.662,Z 624.175,A -85,B 0,C 180,E1 -11974.224,E2 -11974.224} C_VEL
LIN {X 0,Y 381.693,Z 620.602,A -85,B 0,C 180,E1 -11976.127,E2 -11976.127} C_VEL
LIN {X 0,Y 381.937,Z 615.822,A -85,B 0,C 180,E1 -11977.933,E2 -11977.933} C_VEL
LIN {X 0,Y 382.36,Z 609.306,A -85,B 0,C 180,E1 -11979.789,E2 -11979.789} C_VEL
LIN {X 0,Y 382.939,Z 602.298,A -85,B 0,C 180,E1 -11981.379,E2 -11981.379} C_VEL
LIN {X 0,Y 383.776,Z 593.736,A -85,B 0,C 180,E1 -11982.964,E2 -11982.964} C_VEL
LIN {X 0,Y 384.666,Z 584.667,A -85,B 0,C 180,E1 -11984.336,E2 -11984.336} C_VEL
LIN {X 0,Y 385.966,Z 573.516,A -85,B 0,C 180,E1 -11985.716,E2 -11985.716} C_VEL
LIN {X 0,Y 387.102,Z 563.291,A -85,B 0,C 180,E1 -11986.752,E2 -11986.752} C_VEL
LIN {X 0,Y 387.757,Z 555.745,A -85,B 0,C 180,E1 -11987.401,E2 -11987.401} C_VEL
LIN {X 0,Y 387.219,Z 542.174,A -85,B 0,C 180,E1 -11988.477,E2 -11988.477} C_VEL
LIN {X 0,Y 385.511,Z 530.077,A -85,B 0,C 180,E1 -11989.325,E2 -11989.325} C_VEL
LIN {X 0,Y 382.834,Z 518.742,A -85,B 0,C 180,E1 -11990.068,E2 -11990.068} C_VEL
LIN {X 0,Y 382.464,Z 516.486,A -85,B 0,C 180,E1 -11990.23,E2 -11990.23} C_VEL
LIN {X 0,Y 382.932,Z 508.781,A -85,B 0,C 180,E1 -11993.814,E2 -11993.814} C_VEL
LIN {X 0,Y 383.556,Z 501.826,A -85,B 0,C 180,E1 -11997.264,E2 -11997.264} C_VEL
LIN {X 0,Y 384.248,Z 496.405,A -85,B 0,C 180,E1 -12000.178,E2 -12000.178} C_VEL
LIN {X 0,Y 385.025,Z 491.301,A -85,B 0,C 180,E1 -12003.203,E2 -12003.203} C_VEL
LIN {X 0,Y 385.577,Z 487.602,A -85,B 0,C 180,E1 -12005.681,E2 -12005.681} C_VEL
LIN {X 0,Y 385.743,Z 485.901,A -85,B 0,C 180,E1 -12006.959,E2 -12006.959} C_VEL
LIN {X 0,Y 385.677,Z 484.182,A -85,B 0,C 180,E1 -12008.412,E2 -12008.412} C_VEL
LIN {X 0,Y 385.196,Z 481.143,A -85,B 0,C 180,E1 -12011.578,E2 -12011.578} C_VEL
LIN {X 0,Y 384.825,Z 479.04,A -85,B 0,C 180,E1 -12014.582,E2 -12014.582} C_VEL
LIN {X 0,Y 384.587,Z 477.73,A -85,B 0,C 180,E1 -12017.457,E2 -12017.457} C_VEL
LIN {X 0,Y 384.373,Z 477.075,A -85,B 0,C 180,E1 -12020.212,E2 -12020.212} C_VEL
LIN {X 0,Y 384.25,Z 476.956,A -85,B 0,C 180,E1 -12023.588,E2 -12023.588} C_VEL
LIN {X 0,Y 383.928,Z 477.492,A -85,B 0,C 180,E1 -12026.69,E2 -12026.69} C_VEL
LIN {X 0,Y 383.632,Z 478.356,A -85,B 0,C 180,E1 -12029.432,E2 -12029.432} C_VEL
LIN {X 0,Y 383.22,Z 479.79,A -85,B 0,C 180,E1 -12032.711,E2 -12032.711} C_VEL
LIN {X 0,Y 382.929,Z 481.667,A -85,B 0,C 180,E1 -12036.186,E2 -12036.186} C_VEL
LIN {X 0,Y 382.709,Z 484.076,A -85,B 0,C 180,E1 -12039.983,E2 -12039.983} C_VEL
LIN {X 0,Y 383.889,Z 487.251,A -85,B 0,C 180,E1 -12040.241,E2 -12040.241} C_VEL
LIN {X 0,Y 387.824,Z 498.174,A -85,B 0,C 180,E1 -12041.168,E2 -12041.168} C_VEL
LIN {X 0,Y 390.025,Z 506.66,A -85,B 0,C 180,E1 -12041.923,E2 -12041.923} C_VEL
LIN {X 0,Y 389.092,Z 519.602,A -85,B 0,C 180,E1 -12042.932,E2 -12042.932} C_VEL
LIN {X 0,Y 387.955,Z 530.742,A -85,B 0,C 180,E1 -12044.024,E2 -12044.024} C_VEL
LIN {X 0,Y 386.722,Z 541.021,A -85,B 0,C 180,E1 -12045.261,E2 -12045.261} C_VEL
LIN {X 0,Y 385.675,Z 549.862,A -85,B 0,C 180,E1 -12046.565,E2 -12046.565} C_VEL
LIN {X 0,Y 384.633,Z 558.519,A -85,B 0,C 180,E1 -12048.138,E2 -12048.138} C_VEL
LIN {X 0,Y 383.858,Z 565.557,A -85,B 0,C 180,E1 -12049.717,E2 -12049.717} C_VEL
LIN {X 0,Y 383.314,Z 570.338,A -85,B 0,C 180,E1 -12051.034,E2 -12051.034} C_VEL
LIN {X 0,Y 382.73,Z 574.975,A -85,B 0,C 180,E1 -12052.615,E2 -12052.615} C_VEL
LIN {X 0,Y 382.377,Z 577.475,A -85,B 0,C 180,E1 -12053.669,E2 -12053.669} C_VEL
LIN {X 0,Y 382.266,Z 579.466,A -85,B 0,C 180,E1 -12054.726,E2 -12054.726} C_VEL
LIN {X 0,Y 382.191,Z 581.026,A -85,B 0,C 180,E1 -12055.782,E2 -12055.782} C_VEL
LIN {X 0,Y 382.008,Z 582.197,A -85,B 0,C 180,E1 -12056.836,E2 -12056.836} C_VEL
LIN {X 0,Y 381.893,Z 582.954,A -85,B 0,C 180,E1 -12057.891,E2 -12057.891} C_VEL
LIN {X 0,Y 381.794,Z 583.266,A -85,B 0,C 180,E1 -12058.945,E2 -12058.945} C_VEL
LIN {X 0,Y 381.739,Z 583.18,A -85,B 0,C 180,E1 -12060,E2 -12060} C_VEL
LIN {X 0,Y 381.747,Z 582.697,A -85,B 0,C 180,E1 -12061.055,E2 -12061.055} C_VEL
LIN {X 0,Y 381.836,Z 581.785,A -85,B 0,C 180,E1 -12062.11,E2 -12062.11} C_VEL
LIN {X 0,Y 381.886,Z 580.439,A -85,B 0,C 180,E1 -12063.165,E2 -12063.165} C_VEL
LIN {X 0,Y 381.928,Z 577.632,A -85,B 0,C 180,E1 -12064.75,E2 -12064.75} C_VEL
LIN {X 0,Y 382.172,Z 573.779,A -85,B 0,C 180,E1 -12066.335,E2 -12066.335} C_VEL
LIN {X 0,Y 382.43,Z 568.78,A -85,B 0,C 180,E1 -12067.923,E2 -12067.923} C_VEL
LIN {X 0,Y 382.896,Z 562.497,A -85,B 0,C 180,E1 -12069.509,E2 -12069.509} C_VEL
LIN {X 0,Y 383.463,Z 554.714,A -85,B 0,C 180,E1 -12071.096,E2 -12071.096} C_VEL
LIN {X 0,Y 384.187,Z 544.983,A -85,B 0,C 180,E1 -12072.681,E2 -12072.681} C_VEL
LIN {X 0,Y 385.01,Z 535.04,A -85,B 0,C 180,E1 -12073.997,E2 -12073.997} C_VEL
LIN {X 0,Y 385.659,Z 524.731,A -85,B 0,C 180,E1 -12075.109,E2 -12075.109} C_VEL
LIN {X 0,Y 386.401,Z 513.282,A -85,B 0,C 180,E1 -12076.104,E2 -12076.104} C_VEL
LIN {X 0,Y 386.955,Z 502.925,A -85,B 0,C 180,E1 -12076.826,E2 -12076.826} C_VEL
LIN {X 0,Y 384.667,Z 491.669,A -85,B 0,C 180,E1 -12077.543,E2 -12077.543} C_VEL
LIN {X 0,Y 381.903,Z 478.925,A -85,B 0,C 180,E1 -12078.194,E2 -12078.194} C_VEL
LIN {X 0,Y 381.947,Z 475.455,A -85,B 0,C 180,E1 -12081.593,E2 -12081.593} C_VEL
LIN {X 0,Y 382.042,Z 472.023,A -85,B 0,C 180,E1 -12085.031,E2 -12085.031} C_VEL
LIN {X 0,Y 382.172,Z 469.104,A -85,B 0,C 180,E1 -12088.029,E2 -12088.029} C_VEL
LIN {X 0,Y 382.44,Z 468.846,A -85,B 0,C 180,E1 -12090.968,E2 -12090.968} C_VEL
LIN {X 0,Y 382.811,Z 468.801,A -85,B 0,C 180,E1 -12094.69,E2 -12094.69} C_VEL
LIN {X 0,Y 382.982,Z 468.777,A -85,B 0,C 180,E1 -12097.271,E2 -12097.271} C_VEL
LIN {X 0,Y 383.012,Z 468.776,A -85,B 0,C 180,E1 -12099.959,E2 -12099.959} C_VEL
LIN {X 0,Y 383.009,Z 468.776,A -85,B 0,C 180,E1 -12102.779,E2 -12102.779} C_VEL
LIN {X 0,Y 383.001,Z 468.776,A -85,B 0,C 180,E1 -12105.789,E2 -12105.789} C_VEL
LIN {X 0,Y 382.993,Z 468.777,A -85,B 0,C 180,E1 -12108.796,E2 -12108.796} C_VEL
LIN {X 0,Y 383.006,Z 468.778,A -85,B 0,C 180,E1 -12112.096,E2 -12112.096} C_VEL
LIN {X 0,Y 383.023,Z 468.772,A -85,B 0,C 180,E1 -12115.332,E2 -12115.332} C_VEL
LIN {X 0,Y 382.988,Z 468.776,A -85,B 0,C 180,E1 -12119.082,E2 -12119.082} C_VEL
LIN {X 0,Y 383.062,Z 468.769,A -85,B 0,C 180,E1 -12122.698,E2 -12122.698} C_VEL
LIN {X 0,Y 383.058,Z 468.768,A -85,B 0,C 180,E1 -12125.04,E2 -12125.04} C_VEL
LIN {X 0,Y 382.999,Z 468.777,A -85,B 0,C 180,E1 -12128.469,E2 -12128.469} C_VEL
LIN {X 0,Y 383.095,Z 468.767,A -85,B 0,C 180,E1 -12131.828,E2 -12131.828} C_VEL
LIN {X 0,Y 383.116,Z 468.76,A -85,B 0,C 180,E1 -12135.118,E2 -12135.118} C_VEL
LIN {X 0,Y 383.103,Z 468.766,A -85,B 0,C 180,E1 -12138.358,E2 -12138.358} C_VEL
LIN {X 0,Y 383.266,Z 468.746,A -85,B 0,C 180,E1 -12141.979,E2 -12141.979} C_VEL
LIN {X 0,Y 383.201,Z 468.751,A -85,B 0,C 180,E1 -12144.738,E2 -12144.738} C_VEL
LIN {X 0,Y 383.391,Z 468.73,A -85,B 0,C 180,E1 -12147.899,E2 -12147.899} C_VEL
LIN {X 0,Y 383.523,Z 468.714,A -85,B 0,C 180,E1 -12150,E2 -12150} C_VEL
LIN {X 0,Y 383.251,Z 468.744,A -85,B 0,C 180,E1 -12153.153,E2 -12153.153} C_VEL
LIN {X 0,Y 383.268,Z 468.744,A -85,B 0,C 180,E1 -12156.316,E2 -12156.316} C_VEL
LIN {X 0,Y 383.156,Z 468.758,A -85,B 0,C 180,E1 -12159.502,E2 -12159.502} C_VEL
LIN {X 0,Y 383.13,Z 468.76,A -85,B 0,C 180,E1 -12163.536,E2 -12163.536} C_VEL
LIN {X 0,Y 383.099,Z 468.765,A -85,B 0,C 180,E1 -12167.454,E2 -12167.454} C_VEL
LIN {X 0,Y 383.033,Z 468.77,A -85,B 0,C 180,E1 -12170.647,E2 -12170.647} C_VEL
LIN {X 0,Y 383.037,Z 468.774,A -85,B 0,C 180,E1 -12173.807,E2 -12173.807} C_VEL
LIN {X 0,Y 383.05,Z 468.768,A -85,B 0,C 180,E1 -12176.803,E2 -12176.803} C_VEL
LIN {X 0,Y 383.001,Z 468.776,A -85,B 0,C 180,E1 -12180.407,E2 -12180.407} C_VEL
LIN {X 0,Y 382.976,Z 468.777,A -85,B 0,C 180,E1 -12181.37,E2 -12181.37} C_VEL
LIN {X 0,Y 382.316,Z 468.863,A -85,B 0,C 180,E1 -12182.249,E2 -12182.249} C_VEL
LIN {X 0,Y 379.463,Z 469.219,A -85,B 0,C 180,E1 -12183.677,E2 -12183.677} C_VEL
LIN {X 0,Y 377.051,Z 469.517,A -85,B 0,C 180,E1 -12184.831,E2 -12184.831} C_VEL
LIN {X 0,Y 376.026,Z 469.648,A -85,B 0,C 180,E1 -12185.724,E2 -12185.724} C_VEL
LIN {X 0,Y 375.948,Z 469.652,A -85,B 0,C 180,E1 -12186.027,E2 -12186.027} C_VEL
LIN {X 0,Y 375.966,Z 469.654,A -85,B 0,C 180,E1 -12189.462,E2 -12189.462} C_VEL
LIN {X 0,Y 375.937,Z 469.655,A -85,B 0,C 180,E1 -12193.189,E2 -12193.189} C_VEL
LIN {X 0,Y 375.936,Z 469.655,A -85,B 0,C 180,E1 -12196.81,E2 -12196.81} C_VEL
LIN {X 0,Y 375.963,Z 469.651,A -85,B 0,C 180,E1 -12200.537,E2 -12200.537} C_VEL
LIN {X 0,Y 375.966,Z 469.655,A -85,B 0,C 180,E1 -12203.495,E2 -12203.495} C_VEL
LIN {X 0,Y 375.964,Z 469.655,A -85,B 0,C 180,E1 -12205.888,E2 -12205.888} C_VEL
LIN {X 0,Y 375.966,Z 469.655,A -85,B 0,C 180,E1 -12209.687,E2 -12209.687} C_VEL
LIN {X 0,Y 375.997,Z 469.649,A -85,B 0,C 180,E1 -12212.141,E2 -12212.141} C_VEL
LIN {X 0,Y 376.008,Z 469.645,A -85,B 0,C 180,E1 -12214.539,E2 -12214.539} C_VEL
LIN {X 0,Y 375.965,Z 469.654,A -85,B 0,C 180,E1 -12218.045,E2 -12218.045} C_VEL
LIN {X 0,Y 376.025,Z 469.648,A -85,B 0,C 180,E1 -12221.474,E2 -12221.474} C_VEL
LIN {X 0,Y 376.06,Z 469.64,A -85,B 0,C 180,E1 -12224.832,E2 -12224.832} C_VEL
LIN {X 0,Y 376.051,Z 469.641,A -85,B 0,C 180,E1 -12228.136,E2 -12228.136} C_VEL
LIN {X 0,Y 376.258,Z 469.618,A -85,B 0,C 180,E1 -12231.877,E2 -12231.877} C_VEL
LIN {X 0,Y 376.172,Z 469.625,A -85,B 0,C 180,E1 -12234.64,E2 -12234.64} C_VEL
LIN {X 0,Y 376.355,Z 469.606,A -85,B 0,C 180,E1 -12237.859,E2 -12237.859} C_VEL
LIN {X 0,Y 376.49,Z 469.588,A -85,B 0,C 180,E1 -12240,E2 -12240} C_VEL
LIN {X 0,Y 376.186,Z 469.626,A -85,B 0,C 180,E1 -12243.213,E2 -12243.213} C_VEL
LIN {X 0,Y 376.247,Z 469.616,A -85,B 0,C 180,E1 -12246.435,E2 -12246.435} C_VEL
LIN {X 0,Y 376.206,Z 469.621,A -85,B 0,C 180,E1 -12248.595,E2 -12248.595} C_VEL
LIN {X 0,Y 376.051,Z 469.643,A -85,B 0,C 180,E1 -12251.863,E2 -12251.863} C_VEL
LIN {X 0,Y 376.059,Z 469.643,A -85,B 0,C 180,E1 -12255.167,E2 -12255.167} C_VEL
LIN {X 0,Y 376.009,Z 469.645,A -85,B 0,C 180,E1 -12258.527,E2 -12258.527} C_VEL
LIN {X 0,Y 375.963,Z 469.653,A -85,B 0,C 180,E1 -12261.954,E2 -12261.954} C_VEL
LIN {X 0,Y 376.007,Z 469.65,A -85,B 0,C 180,E1 -12265.461,E2 -12265.461} C_VEL
LIN {X 0,Y 375.961,Z 469.655,A -85,B 0,C 180,E1 -12269.08,E2 -12269.08} C_VEL
LIN {X 0,Y 375.951,Z 469.654,A -85,B 0,C 180,E1 -12272.828,E2 -12272.828} C_VEL
LIN {X 0,Y 375.958,Z 469.656,A -85,B 0,C 180,E1 -12275.415,E2 -12275.415} C_VEL
LIN {X 0,Y 375.976,Z 469.649,A -85,B 0,C 180,E1 -12278.271,E2 -12278.271} C_VEL
LIN {X 0,Y 375.988,Z 469.652,A -85,B 0,C 180,E1 -12281.61,E2 -12281.61} C_VEL
LIN {X 0,Y 375.972,Z 469.659,A -85,B 0,C 180,E1 -12285.262,E2 -12285.262} C_VEL
LIN {X 0,Y 376.013,Z 469.77,A -85,B 0,C 180,E1 -12286.154,E2 -12286.154} C_VEL
LIN {X 0,Y 377.155,Z 476.166,A -85,B 0,C 180,E1 -12289.818,E2 -12289.818} C_VEL
LIN {X 0,Y 378.122,Z 482.119,A -85,B 0,C 180,E1 -12293.056,E2 -12293.056} C_VEL
LIN {X 0,Y 378.096,Z 485.659,A -85,B 0,C 180,E1 -12294.872,E2 -12294.872} C_VEL
LIN {X 0,Y 377.415,Z 491.878,A -85,B 0,C 180,E1 -12297.947,E2 -12297.947} C_VEL
LIN {X 0,Y 376.762,Z 498.717,A -85,B 0,C 180,E1 -12301.25,E2 -12301.25} C_VEL
LIN {X 0,Y 376.131,Z 505.712,A -85,B 0,C 180,E1 -12304.548,E2 -12304.548} C_VEL
LIN {X 0,Y 375.501,Z 514.445,A -85,B 0,C 180,E1 -12308.595,E2 -12308.595} C_VEL
LIN {X 0,Y 375.183,Z 520.817,A -85,B 0,C 180,E1 -12311.486,E2 -12311.486} C_VEL
LIN {X 0,Y 376.913,Z 534.49,A -85,B 0,C 180,E1 -12312.085,E2 -12312.085} C_VEL
LIN {X 0,Y 378.473,Z 547.269,A -85,B 0,C 180,E1 -12312.855,E2 -12312.855} C_VEL
LIN {X 0,Y 379.066,Z 555.304,A -85,B 0,C 180,E1 -12313.438,E2 -12313.438} C_VEL
LIN {X 0,Y 378.131,Z 567.74,A -85,B 0,C 180,E1 -12314.504,E2 -12314.504} C_VEL
LIN {X 0,Y 377.249,Z 578.295,A -85,B 0,C 180,E1 -12315.637,E2 -12315.637} C_VEL
LIN {X 0,Y 376.636,Z 587.104,A -85,B 0,C 180,E1 -12316.786,E2 -12316.786} C_VEL
LIN {X 0,Y 375.957,Z 595.702,A -85,B 0,C 180,E1 -12318.134,E2 -12318.134} C_VEL
LIN {X 0,Y 375.312,Z 604.078,A -85,B 0,C 180,E1 -12319.753,E2 -12319.753} C_VEL
LIN {X 0,Y 374.967,Z 610.844,A -85,B 0,C 180,E1 -12321.377,E2 -12321.377} C_VEL
LIN {X 0,Y 374.75,Z 616.23,A -85,B 0,C 180,E1 -12322.998,E2 -12322.998} C_VEL
LIN {X 0,Y 374.666,Z 620.397,A -85,B 0,C 180,E1 -12324.619,E2 -12324.619} C_VEL
LIN {X 0,Y 374.613,Z 622.559,A -85,B 0,C 180,E1 -12325.697,E2 -12325.697} C_VEL
LIN {X 0,Y 374.598,Z 624.228,A -85,B 0,C 180,E1 -12326.774,E2 -12326.774} C_VEL
LIN {X 0,Y 374.711,Z 625.481,A -85,B 0,C 180,E1 -12327.85,E2 -12327.85} C_VEL
LIN {X 0,Y 374.67,Z 626.301,A -85,B 0,C 180,E1 -12328.925,E2 -12328.925} C_VEL
LIN {X 0,Y 374.665,Z 626.656,A -85,B 0,C 180,E1 -12330,E2 -12330} C_VEL
LIN {X 0,Y 374.663,Z 626.59,A -85,B 0,C 180,E1 -12331.075,E2 -12331.075} C_VEL
LIN {X 0,Y 374.67,Z 626.115,A -85,B 0,C 180,E1 -12332.15,E2 -12332.15} C_VEL
LIN {X 0,Y 374.553,Z 625.215,A -85,B 0,C 180,E1 -12333.227,E2 -12333.227} C_VEL
LIN {X 0,Y 374.585,Z 623.857,A -85,B 0,C 180,E1 -12334.304,E2 -12334.304} C_VEL
LIN {X 0,Y 374.589,Z 620.694,A -85,B 0,C 180,E1 -12336.077,E2 -12336.077} C_VEL
LIN {X 0,Y 374.875,Z 615.629,A -85,B 0,C 180,E1 -12338.083,E2 -12338.083} C_VEL
LIN {X 0,Y 375.332,Z 609.216,A -85,B 0,C 180,E1 -12339.974,E2 -12339.974} C_VEL
LIN {X 0,Y 375.97,Z 602.308,A -85,B 0,C 180,E1 -12341.593,E2 -12341.593} C_VEL
LIN {X 0,Y 376.844,Z 593.87,A -85,B 0,C 180,E1 -12343.207,E2 -12343.207} C_VEL
LIN {X 0,Y 377.803,Z 585.005,A -85,B 0,C 180,E1 -12344.603,E2 -12344.603} C_VEL
LIN {X 0,Y 379.166,Z 574.056,A -85,B 0,C 180,E1 -12346.005,E2 -12346.005} C_VEL
LIN {X 0,Y 380.534,Z 562.745,A -85,B 0,C 180,E1 -12347.188,E2 -12347.188} C_VEL
LIN {X 0,Y 381.029,Z 555.3,A -85,B 0,C 180,E1 -12347.857,E2 -12347.857} C_VEL
LIN {X 0,Y 380.493,Z 541.521,A -85,B 0,C 180,E1 -12348.988,E2 -12348.988} C_VEL
LIN {X 0,Y 378.956,Z 530.878,A -85,B 0,C 180,E1 -12349.784,E2 -12349.784} C_VEL
LIN {X 0,Y 375.934,Z 518.33,A -85,B 0,C 180,E1 -12350.673,E2 -12350.673} C_VEL
LIN {X 0,Y 375.481,Z 515.915,A -85,B 0,C 180,E1 -12350.832,E2 -12350.832} C_VEL
LIN {X 0,Y 375.961,Z 508.726,A -85,B 0,C 180,E1 -12354.284,E2 -12354.284} C_VEL
LIN {X 0,Y 376.65,Z 501.895,A -85,B 0,C 180,E1 -12357.806,E2 -12357.806} C_VEL
LIN {X 0,Y 377.436,Z 496.095,A -85,B 0,C 180,E1 -12361.07,E2 -12361.07} C_VEL
LIN {X 0,Y 378.209,Z 491.601,A -85,B 0,C 180,E1 -12363.881,E2 -12363.881} C_VEL
LIN {X 0,Y 378.724,Z 488.029,A -85,B 0,C 180,E1 -12366.429,E2 -12366.429} C_VEL
LIN {X 0,Y 378.674,Z 485.277,A -85,B 0,C 180,E1 -12368.785,E2 -12368.785} C_VEL
LIN {X 0,Y 378.21,Z 482.361,A -85,B 0,C 180,E1 -12371.987,E2 -12371.987} C_VEL
LIN {X 0,Y 377.868,Z 480.358,A -85,B 0,C 180,E1 -12375.028,E2 -12375.028} C_VEL
LIN {X 0,Y 377.607,Z 479.067,A -85,B 0,C 180,E1 -12378.115,E2 -12378.115} C_VEL
LIN {X 0,Y 377.404,Z 478.44,A -85,B 0,C 180,E1 -12381.456,E2 -12381.456} C_VEL
LIN {X 0,Y 377.325,Z 478.412,A -85,B 0,C 180,E1 -12383.414,E2 -12383.414} C_VEL
LIN {X 0,Y 376.942,Z 478.971,A -85,B 0,C 180,E1 -12387.037,E2 -12387.037} C_VEL
LIN {X 0,Y 376.6,Z 479.805,A -85,B 0,C 180,E1 -12389.744,E2 -12389.744} C_VEL
LIN {X 0,Y 376.156,Z 481.36,A -85,B 0,C 180,E1 -12393.358,E2 -12393.358} C_VEL
LIN {X 0,Y 375.856,Z 483.254,A -85,B 0,C 180,E1 -12396.879,E2 -12396.879} C_VEL
LIN {X 0,Y 375.739,Z 484.775,A -85,B 0,C 180,E1 -12399.359,E2 -12399.359} C_VEL
LIN {X 0,Y 376.816,Z 487.746,A -85,B 0,C 180,E1 -12399.611,E2 -12399.611} C_VEL
LIN {X 0,Y 380.882,Z 498.384,A -85,B 0,C 180,E1 -12400.602,E2 -12400.602} C_VEL
LIN {X 0,Y 383.59,Z 508.364,A -85,B 0,C 180,E1 -12401.534,E2 -12401.534} C_VEL
LIN {X 0,Y 382.642,Z 520.243,A -85,B 0,C 180,E1 -12402.497,E2 -12402.497} C_VEL
LIN {X 0,Y 381.442,Z 531.06,A -85,B 0,C 180,E1 -12403.586,E2 -12403.586} C_VEL
LIN {X 0,Y 379.994,Z 542.462,A -85,B 0,C 180,E1 -12404.994,E2 -12404.994} C_VEL
LIN {X 0,Y 378.881,Z 551.112,A -85,B 0,C 180,E1 -12406.32,E2 -12406.32} C_VEL
LIN {X 0,Y 377.797,Z 559.603,A -85,B 0,C 180,E1 -12407.92,E2 -12407.92} C_VEL
LIN {X 0,Y 376.934,Z 566.487,A -85,B 0,C 180,E1 -12409.526,E2 -12409.526} C_VEL
LIN {X 0,Y 376.363,Z 571.172,A -85,B 0,C 180,E1 -12410.867,E2 -12410.867} C_VEL
LIN {X 0,Y 375.721,Z 575.738,A -85,B 0,C 180,E1 -12412.476,E2 -12412.476} C_VEL
LIN {X 0,Y 375.36,Z 578.189,A -85,B 0,C 180,E1 -12413.55,E2 -12413.55} C_VEL
LIN {X 0,Y 375.232,Z 580.12,A -85,B 0,C 180,E1 -12414.627,E2 -12414.627} C_VEL
LIN {X 0,Y 375.15,Z 581.636,A -85,B 0,C 180,E1 -12415.703,E2 -12415.703} C_VEL
LIN {X 0,Y 374.958,Z 582.762,A -85,B 0,C 180,E1 -12416.777,E2 -12416.777} C_VEL
LIN {X 0,Y 374.829,Z 583.45,A -85,B 0,C 180,E1 -12417.851,E2 -12417.851} C_VEL
LIN {X 0,Y 374.724,Z 583.721,A -85,B 0,C 180,E1 -12418.926,E2 -12418.926} C_VEL
LIN {X 0,Y 374.667,Z 583.6,A -85,B 0,C 180,E1 -12420,E2 -12420} C_VEL
LIN {X 0,Y 374.679,Z 583.079,A -85,B 0,C 180,E1 -12421.075,E2 -12421.075} C_VEL
LIN {X 0,Y 374.772,Z 582.105,A -85,B 0,C 180,E1 -12422.15,E2 -12422.15} C_VEL
LIN {X 0,Y 374.793,Z 580.72,A -85,B 0,C 180,E1 -12423.225,E2 -12423.225} C_VEL
LIN {X 0,Y 374.866,Z 577.835,A -85,B 0,C 180,E1 -12424.84,E2 -12424.84} C_VEL
LIN {X 0,Y 375.106,Z 573.898,A -85,B 0,C 180,E1 -12426.455,E2 -12426.455} C_VEL
LIN {X 0,Y 375.369,Z 568.808,A -85,B 0,C 180,E1 -12428.073,E2 -12428.073} C_VEL
LIN {X 0,Y 375.865,Z 562.424,A -85,B 0,C 180,E1 -12429.688,E2 -12429.688} C_VEL
LIN {X 0,Y 376.449,Z 554.484,A -85,B 0,C 180,E1 -12431.305,E2 -12431.305} C_VEL
LIN {X 0,Y 377.218,Z 544.618,A -85,B 0,C 180,E1 -12432.919,E2 -12432.919} C_VEL
LIN {X 0,Y 378.066,Z 534.582,A -85,B 0,C 180,E1 -12434.247,E2 -12434.247} C_VEL
LIN {X 0,Y 378.821,Z 523.168,A -85,B 0,C 180,E1 -12435.467,E2 -12435.467} C_VEL
LIN {X 0,Y 379.627,Z 510.548,A -85,B 0,C 180,E1 -12436.537,E2 -12436.537} C_VEL
LIN {X 0,Y 379.982,Z 503.757,A -85,B 0,C 180,E1 -12437.006,E2 -12437.006} C_VEL
LIN {X 0,Y 377.511,Z 491.792,A -85,B 0,C 180,E1 -12437.785,E2 -12437.785} C_VEL
LIN {X 0,Y 374.848,Z 479.296,A -85,B 0,C 180,E1 -12438.429,E2 -12438.429} C_VEL
LIN {X 0,Y 374.847,Z 476.816,A -85,B 0,C 180,E1 -12440.869,E2 -12440.869} C_VEL
LIN {X 0,Y 374.937,Z 473.349,A -85,B 0,C 180,E1 -12444.355,E2 -12444.355} C_VEL
LIN {X 0,Y 375.112,Z 469.88,A -85,B 0,C 180,E1 -12447.931,E2 -12447.931} C_VEL
LIN {X 0,Y 375.444,Z 469.717,A -85,B 0,C 180,E1 -12451.611,E2 -12451.611} C_VEL
LIN {X 0,Y 375.791,Z 469.676,A -85,B 0,C 180,E1 -12454.625,E2 -12454.625} C_VEL
LIN {X 0,Y 375.92,Z 469.659,A -85,B 0,C 180,E1 -12456.746,E2 -12456.746} C_VEL
LIN {X 0,Y 375.992,Z 469.65,A -85,B 0,C 180,E1 -12459.971,E2 -12459.971} C_VEL
LIN {X 0,Y 375.934,Z 469.657,A -85,B 0,C 180,E1 -12463.766,E2 -12463.766} C_VEL
LIN {X 0,Y 375.938,Z 469.655,A -85,B 0,C 180,E1 -12466.811,E2 -12466.811} C_VEL
LIN {X 0,Y 375.968,Z 469.654,A -85,B 0,C 180,E1 -12470.538,E2 -12470.538} C_VEL
LIN {X 0,Y 375.969,Z 469.65,A -85,B 0,C 180,E1 -12473.495,E2 -12473.495} C_VEL
LIN {X 0,Y 375.967,Z 469.654,A -85,B 0,C 180,E1 -12475.889,E2 -12475.889} C_VEL
LIN {X 0,Y 375.969,Z 469.652,A -85,B 0,C 180,E1 -12479.687,E2 -12479.687} C_VEL
LIN {X 0,Y 376.025,Z 469.644,A -85,B 0,C 180,E1 -12483.348,E2 -12483.348} C_VEL
LIN {X 0,Y 376.002,Z 469.646,A -85,B 0,C 180,E1 -12486.888,E2 -12486.888} C_VEL
LIN {X 0,Y 376.004,Z 469.65,A -85,B 0,C 180,E1 -12490.339,E2 -12490.339} C_VEL
LIN {X 0,Y 376.035,Z 469.645,A -85,B 0,C 180,E1 -12493.719,E2 -12493.719} C_VEL
LIN {X 0,Y 376.109,Z 469.633,A -85,B 0,C 180,E1 -12497.042,E2 -12497.042} C_VEL
LIN {X 0,Y 376.121,Z 469.635,A -85,B 0,C 180,E1 -12500.318,E2 -12500.318} C_VEL
LIN {X 0,Y 376.239,Z 469.619,A -85,B 0,C 180,E1 -12503.565,E2 -12503.565} C_VEL
LIN {X 0,Y 376.357,Z 469.606,A -85,B 0,C 180,E1 -12507.859,E2 -12507.859} C_VEL
LIN {X 0,Y 376.493,Z 469.59,A -85,B 0,C 180,E1 -12510,E2 -12510} C_VEL
LIN {X 0,Y 376.189,Z 469.624,A -85,B 0,C 180,E1 -12513.213,E2 -12513.213} C_VEL
LIN {X 0,Y 376.225,Z 469.62,A -85,B 0,C 180,E1 -12516.435,E2 -12516.435} C_VEL
LIN {X 0,Y 376.124,Z 469.635,A -85,B 0,C 180,E1 -12519.681,E2 -12519.681} C_VEL
LIN {X 0,Y 376.094,Z 469.638,A -85,B 0,C 180,E1 -12523.657,E2 -12523.657} C_VEL
LIN {X 0,Y 376.049,Z 469.644,A -85,B 0,C 180,E1 -12527.607,E2 -12527.607} C_VEL
LIN {X 0,Y 375.982,Z 469.648,A -85,B 0,C 180,E1 -12530.832,E2 -12530.832} C_VEL
LIN {X 0,Y 375.998,Z 469.65,A -85,B 0,C 180,E1 -12534.281,E2 -12534.281} C_VEL
LIN {X 0,Y 376.023,Z 469.644,A -85,B 0,C 180,E1 -12536.652,E2 -12536.652} C_VEL
LIN {X 0,Y 375.968,Z 469.653,A -85,B 0,C 180,E1 -12540.312,E2 -12540.312} C_VEL
LIN {X 0,Y 375.965,Z 469.654,A -85,B 0,C 180,E1 -12544.111,E2 -12544.111} C_VEL
LIN {X 0,Y 375.948,Z 469.652,A -85,B 0,C 180,E1 -12546.027,E2 -12546.027} C_VEL
LIN {X 0,Y 375.301,Z 469.734,A -85,B 0,C 180,E1 -12546.921,E2 -12546.921} C_VEL
LIN {X 0,Y 372.466,Z 470.088,A -85,B 0,C 180,E1 -12548.375,E2 -12548.375} C_VEL
LIN {X 0,Y 370.041,Z 470.393,A -85,B 0,C 180,E1 -12549.551,E2 -12549.551} C_VEL
LIN {X 0,Y 368.979,Z 470.522,A -85,B 0,C 180,E1 -12550.46,E2 -12550.46} C_VEL
LIN {X 0,Y 368.882,Z 470.532,A -85,B 0,C 180,E1 -12550.768,E2 -12550.768} C_VEL
LIN {X 0,Y 368.886,Z 470.537,A -85,B 0,C 180,E1 -12553.616,E2 -12553.616} C_VEL
LIN {X 0,Y 368.888,Z 470.533,A -85,B 0,C 180,E1 -12556.696,E2 -12556.696} C_VEL
LIN {X 0,Y 368.914,Z 470.534,A -85,B 0,C 180,E1 -12559.642,E2 -12559.642} C_VEL
LIN {X 0,Y 368.904,Z 470.532,A -85,B 0,C 180,E1 -12563.144,E2 -12563.144} C_VEL
LIN {X 0,Y 368.9,Z 470.531,A -85,B 0,C 180,E1 -12566.462,E2 -12566.462} C_VEL
LIN {X 0,Y 368.93,Z 470.528,A -85,B 0,C 180,E1 -12569.046,E2 -12569.046} C_VEL
LIN {X 0,Y 368.981,Z 470.525,A -85,B 0,C 180,E1 -12571.564,E2 -12571.564} C_VEL
LIN {X 0,Y 369.001,Z 470.52,A -85,B 0,C 180,E1 -12574.019,E2 -12574.019} C_VEL
LIN {X 0,Y 368.934,Z 470.531,A -85,B 0,C 180,E1 -12577.605,E2 -12577.605} C_VEL
LIN {X 0,Y 368.984,Z 470.522,A -85,B 0,C 180,E1 -12581.107,E2 -12581.107} C_VEL
LIN {X 0,Y 368.999,Z 470.519,A -85,B 0,C 180,E1 -12584.535,E2 -12584.535} C_VEL
LIN {X 0,Y 369.006,Z 470.52,A -85,B 0,C 180,E1 -12587.906,E2 -12587.906} C_VEL
LIN {X 0,Y 369.23,Z 470.494,A -85,B 0,C 180,E1 -12591.8,E2 -12591.8} C_VEL
LIN {X 0,Y 369.145,Z 470.5,A -85,B 0,C 180,E1 -12594.537,E2 -12594.537} C_VEL
LIN {X 0,Y 369.32,Z 470.482,A -85,B 0,C 180,E1 -12597.819,E2 -12597.819} C_VEL
LIN {X 0,Y 369.459,Z 470.463,A -85,B 0,C 180,E1 -12600,E2 -12600} C_VEL
LIN {X 0,Y 369.317,Z 470.479,A -85,B 0,C 180,E1 -12602.181,E2 -12602.181} C_VEL
LIN {X 0,Y 369.209,Z 470.493,A -85,B 0,C 180,E1 -12606.558,E2 -12606.558} C_VEL
LIN {X 0,Y 369.138,Z 470.502,A -85,B 0,C 180,E1 -12608.761,E2 -12608.761} C_VEL
LIN {X 0,Y 369.006,Z 470.519,A -85,B 0,C 180,E1 -12612.093,E2 -12612.093} C_VEL
LIN {X 0,Y 368.998,Z 470.523,A -85,B 0,C 180,E1 -12615.465,E2 -12615.465} C_VEL
LIN {X 0,Y 368.958,Z 470.525,A -85,B 0,C 180,E1 -12618.894,E2 -12618.894} C_VEL
LIN {X 0,Y 368.932,Z 470.527,A -85,B 0,C 180,E1 -12622.395,E2 -12622.395} C_VEL
LIN {X 0,Y 369,Z 470.519,A -85,B 0,C 180,E1 -12625.98,E2 -12625.98} C_VEL
LIN {X 0,Y 368.915,Z 470.532,A -85,B 0,C 180,E1 -12629.69,E2 -12629.69} C_VEL
LIN {X 0,Y 368.898,Z 470.534,A -85,B 0,C 180,E1 -12633.044,E2 -12633.044} C_VEL
LIN {X 0,Y 368.918,Z 470.529,A -85,B 0,C 180,E1 -12636.197,E2 -12636.197} C_VEL
LIN {X 0,Y 368.906,Z 470.533,A -85,B 0,C 180,E1 -12638.953,E2 -12638.953} C_VEL
LIN {X 0,Y 368.941,Z 470.527,A -85,B 0,C 180,E1 -12642.02,E2 -12642.02} C_VEL
LIN {X 0,Y 368.926,Z 470.537,A -85,B 0,C 180,E1 -12645.183,E2 -12645.183} C_VEL
LIN {X 0,Y 368.975,Z 470.594,A -85,B 0,C 180,E1 -12645.885,E2 -12645.885} C_VEL
LIN {X 0,Y 370.034,Z 476.659,A -85,B 0,C 180,E1 -12649.439,E2 -12649.439} C_VEL
LIN {X 0,Y 371.014,Z 482.536,A -85,B 0,C 180,E1 -12652.711,E2 -12652.711} C_VEL
LIN {X 0,Y 371.092,Z 485.967,A -85,B 0,C 180,E1 -12654.525,E2 -12654.525} C_VEL
LIN {X 0,Y 370.53,Z 491.39,A -85,B 0,C 180,E1 -12657.278,E2 -12657.278} C_VEL
LIN {X 0,Y 369.756,Z 498.849,A -85,B 0,C 180,E1 -12660.966,E2 -12660.966} C_VEL
LIN {X 0,Y 369.049,Z 506.446,A -85,B 0,C 180,E1 -12664.629,E2 -12664.629} C_VEL
LIN {X 0,Y 368.467,Z 513.903,A -85,B 0,C 180,E1 -12668.165,E2 -12668.165} C_VEL
LIN {X 0,Y 368.095,Z 520.445,A -85,B 0,C 180,E1 -12671.223,E2 -12671.223} C_VEL
LIN {X 0,Y 369.819,Z 534.106,A -85,B 0,C 180,E1 -12671.841,E2 -12671.841} C_VEL
LIN {X 0,Y 371.392,Z 547.31,A -85,B 0,C 180,E1 -12672.66,E2 -12672.66} C_VEL
LIN {X 0,Y 371.96,Z 556.989,A -85,B 0,C 180,E1 -12673.395,E2 -12673.395} C_VEL
LIN {X 0,Y 371.031,Z 568.991,A -85,B 0,C 180,E1 -12674.482,E2 -12674.482} C_VEL
LIN {X 0,Y 370.138,Z 579.825,A -85,B 0,C 180,E1 -12675.71,E2 -12675.71} C_VEL
LIN {X 0,Y 369.324,Z 589.597,A -85,B 0,C 180,E1 -12677.08,E2 -12677.08} C_VEL
LIN {X 0,Y 368.713,Z 597.683,A -85,B 0,C 180,E1 -12678.455,E2 -12678.455} C_VEL
LIN {X 0,Y 368.144,Z 605.644,A -85,B 0,C 180,E1 -12680.107,E2 -12680.107} C_VEL
LIN {X 0,Y 367.822,Z 612,A -85,B 0,C 180,E1 -12681.761,E2 -12681.761} C_VEL
LIN {X 0,Y 367.636,Z 617.03,A -85,B 0,C 180,E1 -12683.414,E2 -12683.414} C_VEL
LIN {X 0,Y 367.612,Z 620.888,A -85,B 0,C 180,E1 -12685.065,E2 -12685.065} C_VEL
LIN {X 0,Y 367.511,Z 623.653,A -85,B 0,C 180,E1 -12686.711,E2 -12686.711} C_VEL
LIN {X 0,Y 367.644,Z 624.938,A -85,B 0,C 180,E1 -12687.809,E2 -12687.809} C_VEL
LIN {X 0,Y 367.604,Z 625.79,A -85,B 0,C 180,E1 -12688.905,E2 -12688.905} C_VEL
LIN {X 0,Y 367.595,Z 626.204,A -85,B 0,C 180,E1 -12690,E2 -12690} C_VEL
LIN {X 0,Y 367.596,Z 626.166,A -85,B 0,C 180,E1 -12691.096,E2 -12691.096} C_VEL
LIN {X 0,Y 367.57,Z 625.717,A -85,B 0,C 180,E1 -12692.192,E2 -12692.192} C_VEL
LIN {X 0,Y 367.465,Z 624.854,A -85,B 0,C 180,E1 -12693.29,E2 -12693.29} C_VEL
LIN {X 0,Y 367.51,Z 623.55,A -85,B 0,C 180,E1 -12694.387,E2 -12694.387} C_VEL
LIN {X 0,Y 367.49,Z 620.796,A -85,B 0,C 180,E1 -12696.03,E2 -12696.03} C_VEL
LIN {X 0,Y 367.705,Z 616.983,A -85,B 0,C 180,E1 -12697.689,E2 -12697.689} C_VEL
LIN {X 0,Y 368.064,Z 612.073,A -85,B 0,C 180,E1 -12699.341,E2 -12699.341} C_VEL
LIN {X 0,Y 368.701,Z 604.786,A -85,B 0,C 180,E1 -12701.267,E2 -12701.267} C_VEL
LIN {X 0,Y 369.628,Z 597.023,A -85,B 0,C 180,E1 -12702.91,E2 -12702.91} C_VEL
LIN {X 0,Y 370.561,Z 588.214,A -85,B 0,C 180,E1 -12704.446,E2 -12704.446} C_VEL
LIN {X 0,Y 372.084,Z 576.886,A -85,B 0,C 180,E1 -12706.036,E2 -12706.036} C_VEL
LIN {X 0,Y 373.456,Z 566.35,A -85,B 0,C 180,E1 -12707.242,E2 -12707.242} C_VEL
LIN {X 0,Y 374.399,Z 556.567,A -85,B 0,C 180,E1 -12708.185,E2 -12708.185} C_VEL
LIN {X 0,Y 374.02,Z 543.394,A -85,B 0,C 180,E1 -12709.33,E2 -12709.33} C_VEL
LIN {X 0,Y 372.718,Z 533.302,A -85,B 0,C 180,E1 -12710.144,E2 -12710.144} C_VEL
LIN {X 0,Y 370.08,Z 521.534,A -85,B 0,C 180,E1 -12711.045,E2 -12711.045} C_VEL
LIN {X 0,Y 368.494,Z 515.265,A -85,B 0,C 180,E1 -12711.51,E2 -12711.51} C_VEL
LIN {X 0,Y 369.03,Z 508.719,A -85,B 0,C 180,E1 -12714.77,E2 -12714.77} C_VEL
LIN {X 0,Y 369.743,Z 501.988,A -85,B 0,C 180,E1 -12718.372,E2 -12718.372} C_VEL
LIN {X 0,Y 370.509,Z 496.819,A -85,B 0,C 180,E1 -12721.396,E2 -12721.396} C_VEL
LIN {X 0,Y 371.395,Z 491.941,A -85,B 0,C 180,E1 -12724.59,E2 -12724.59} C_VEL
LIN {X 0,Y 371.822,Z 488.234,A -85,B 0,C 180,E1 -12727.452,E2 -12727.452} C_VEL
LIN {X 0,Y 371.526,Z 485.573,A -85,B 0,C 180,E1 -12730.029,E2 -12730.029} C_VEL
LIN {X 0,Y 371.131,Z 483.193,A -85,B 0,C 180,E1 -12732.979,E2 -12732.979} C_VEL
LIN {X 0,Y 370.85,Z 481.403,A -85,B 0,C 180,E1 -12736.066,E2 -12736.066} C_VEL
LIN {X 0,Y 370.57,Z 480.292,A -85,B 0,C 180,E1 -12739.343,E2 -12739.343} C_VEL
LIN {X 0,Y 370.378,Z 479.888,A -85,B 0,C 180,E1 -12742.841,E2 -12742.841} C_VEL
LIN {X 0,Y 370.146,Z 480.055,A -85,B 0,C 180,E1 -12745.277,E2 -12745.277} C_VEL
LIN {X 0,Y 369.861,Z 480.573,A -85,B 0,C 180,E1 -12747.856,E2 -12747.856} C_VEL
LIN {X 0,Y 369.459,Z 481.63,A -85,B 0,C 180,E1 -12751.049,E2 -12751.049} C_VEL
LIN {X 0,Y 369.117,Z 482.938,A -85,B 0,C 180,E1 -12754.029,E2 -12754.029} C_VEL
LIN {X 0,Y 368.795,Z 484.855,A -85,B 0,C 180,E1 -12757.596,E2 -12757.596} C_VEL
LIN {X 0,Y 368.715,Z 485.491,A -85,B 0,C 180,E1 -12758.676,E2 -12758.676} C_VEL
LIN {X 0,Y 369.992,Z 488.744,A -85,B 0,C 180,E1 -12758.987,E2 -12758.987} C_VEL
LIN {X 0,Y 373.997,Z 498.661,A -85,B 0,C 180,E1 -12759.982,E2 -12759.982} C_VEL
LIN {X 0,Y 377.185,Z 510.069,A -85,B 0,C 180,E1 -12761.13,E2 -12761.13} C_VEL
LIN {X 0,Y 376.258,Z 520.988,A -85,B 0,C 180,E1 -12762.049,E2 -12762.049} C_VEL
LIN {X 0,Y 374.895,Z 532.279,A -85,B 0,C 180,E1 -12763.213,E2 -12763.213} C_VEL
LIN {X 0,Y 373.578,Z 542.066,A -85,B 0,C 180,E1 -12764.45,E2 -12764.45} C_VEL
LIN {X 0,Y 372.276,Z 550.841,A -85,B 0,C 180,E1 -12765.794,E2 -12765.794} C_VEL
LIN {X 0,Y 371.142,Z 559.442,A -85,B 0,C 180,E1 -12767.422,E2 -12767.422} C_VEL
LIN {X 0,Y 370.191,Z 566.444,A -85,B 0,C 180,E1 -12769.056,E2 -12769.056} C_VEL
LIN {X 0,Y 369.417,Z 572.075,A -85,B 0,C 180,E1 -12770.694,E2 -12770.694} C_VEL
LIN {X 0,Y 368.723,Z 576.609,A -85,B 0,C 180,E1 -12772.37,E2 -12772.37} C_VEL
LIN {X 0,Y 368.346,Z 578.883,A -85,B 0,C 180,E1 -12773.427,E2 -12773.427} C_VEL
LIN {X 0,Y 368.183,Z 580.776,A -85,B 0,C 180,E1 -12774.523,E2 -12774.523} C_VEL
LIN {X 0,Y 368.111,Z 582.252,A -85,B 0,C 180,E1 -12775.62,E2 -12775.62} C_VEL
LIN {X 0,Y 367.91,Z 583.329,A -85,B 0,C 180,E1 -12776.715,E2 -12776.715} C_VEL
LIN {X 0,Y 367.767,Z 583.956,A -85,B 0,C 180,E1 -12777.81,E2 -12777.81} C_VEL
LIN {X 0,Y 367.656,Z 584.188,A -85,B 0,C 180,E1 -12778.905,E2 -12778.905} C_VEL
LIN {X 0,Y 367.598,Z 584.023,A -85,B 0,C 180,E1 -12780,E2 -12780} C_VEL
LIN {X 0,Y 367.613,Z 583.438,A -85,B 0,C 180,E1 -12781.096,E2 -12781.096} C_VEL
LIN {X 0,Y 367.691,Z 582.412,A -85,B 0,C 180,E1 -12782.191,E2 -12782.191} C_VEL
LIN {X 0,Y 367.7,Z 580.99,A -85,B 0,C 180,E1 -12783.287,E2 -12783.287} C_VEL
LIN {X 0,Y 367.809,Z 578.03,A -85,B 0,C 180,E1 -12784.933,E2 -12784.933} C_VEL
LIN {X 0,Y 368.059,Z 574.011,A -85,B 0,C 180,E1 -12786.579,E2 -12786.579} C_VEL
LIN {X 0,Y 368.408,Z 567.853,A -85,B 0,C 180,E1 -12788.502,E2 -12788.502} C_VEL
LIN {X 0,Y 368.925,Z 561.089,A -85,B 0,C 180,E1 -12790.15,E2 -12790.15} C_VEL
LIN {X 0,Y 369.563,Z 552.733,A -85,B 0,C 180,E1 -12791.797,E2 -12791.797} C_VEL
LIN {X 0,Y 370.266,Z 544.25,A -85,B 0,C 180,E1 -12793.166,E2 -12793.166} C_VEL
LIN {X 0,Y 371.118,Z 534.253,A -85,B 0,C 180,E1 -12794.487,E2 -12794.487} C_VEL
LIN {X 0,Y 371.903,Z 522.385,A -85,B 0,C 180,E1 -12795.763,E2 -12795.763} C_VEL
LIN {X 0,Y 372.644,Z 511.251,A -85,B 0,C 180,E1 -12796.715,E2 -12796.715} C_VEL
LIN {X 0,Y 373.016,Z 504.512,A -85,B 0,C 180,E1 -12797.192,E2 -12797.192} C_VEL
LIN {X 0,Y 370.158,Z 490.853,A -85,B 0,C 180,E1 -12798.1,E2 -12798.1} C_VEL
LIN {X 0,Y 367.789,Z 479.665,A -85,B 0,C 180,E1 -12798.667,E2 -12798.667} C_VEL
LIN {X 0,Y 367.766,Z 477.026,A -85,B 0,C 180,E1 -12801.29,E2 -12801.29} C_VEL
LIN {X 0,Y 367.907,Z 473.52,A -85,B 0,C 180,E1 -12804.851,E2 -12804.851} C_VEL
LIN {X 0,Y 367.973,Z 471.181,A -85,B 0,C 180,E1 -12807.283,E2 -12807.283} C_VEL
LIN {X 0,Y 368.121,Z 470.634,A -85,B 0,C 180,E1 -12808.572,E2 -12808.572} C_VEL
LIN {X 0,Y 368.466,Z 470.59,A -85,B 0,C 180,E1 -12812.281,E2 -12812.281} C_VEL
LIN {X 0,Y 368.765,Z 470.549,A -85,B 0,C 180,E1 -12814.964,E2 -12814.964} C_VEL
LIN {X 0,Y 368.878,Z 470.534,A -85,B 0,C 180,E1 -12817.567,E2 -12817.567} C_VEL
LIN {X 0,Y 368.915,Z 470.533,A -85,B 0,C 180,E1 -12820.37,E2 -12820.37} C_VEL
LIN {X 0,Y 368.886,Z 470.534,A -85,B 0,C 180,E1 -12823.616,E2 -12823.616} C_VEL
LIN {X 0,Y 368.89,Z 470.534,A -85,B 0,C 180,E1 -12826.696,E2 -12826.696} C_VEL
LIN {X 0,Y 368.916,Z 470.53,A -85,B 0,C 180,E1 -12829.643,E2 -12829.643} C_VEL
LIN {X 0,Y 368.907,Z 470.529,A -85,B 0,C 180,E1 -12833.144,E2 -12833.144} C_VEL
LIN {X 0,Y 368.903,Z 470.534,A -85,B 0,C 180,E1 -12836.462,E2 -12836.462} C_VEL
LIN {X 0,Y 368.934,Z 470.527,A -85,B 0,C 180,E1 -12839.047,E2 -12839.047} C_VEL
LIN {X 0,Y 368.968,Z 470.524,A -85,B 0,C 180,E1 -12842.797,E2 -12842.797} C_VEL
LIN {X 0,Y 368.951,Z 470.529,A -85,B 0,C 180,E1 -12846.113,E2 -12846.113} C_VEL
LIN {X 0,Y 368.942,Z 470.53,A -85,B 0,C 180,E1 -12849.947,E2 -12849.947} C_VEL
LIN {X 0,Y 368.981,Z 470.521,A -85,B 0,C 180,E1 -12853.399,E2 -12853.399} C_VEL
LIN {X 0,Y 369.063,Z 470.511,A -85,B 0,C 180,E1 -12856.79,E2 -12856.79} C_VEL
LIN {X 0,Y 369.07,Z 470.515,A -85,B 0,C 180,E1 -12860.132,E2 -12860.132} C_VEL
LIN {X 0,Y 369.199,Z 470.494,A -85,B 0,C 180,E1 -12863.441,E2 -12863.441} C_VEL
LIN {X 0,Y 369.322,Z 470.482,A -85,B 0,C 180,E1 -12867.819,E2 -12867.819} C_VEL
LIN {X 0,Y 369.462,Z 470.466,A -85,B 0,C 180,E1 -12870,E2 -12870} C_VEL
LIN {X 0,Y 369.322,Z 470.482,A -85,B 0,C 180,E1 -12872.181,E2 -12872.181} C_VEL
LIN {X 0,Y 369.183,Z 470.496,A -85,B 0,C 180,E1 -12876.558,E2 -12876.558} C_VEL
LIN {X 0,Y 369.072,Z 470.514,A -85,B 0,C 180,E1 -12879.868,E2 -12879.868} C_VEL
LIN {X 0,Y 369.042,Z 470.517,A -85,B 0,C 180,E1 -12883.772,E2 -12883.772} C_VEL
LIN {X 0,Y 369.005,Z 470.522,A -85,B 0,C 180,E1 -12887.768,E2 -12887.768} C_VEL
LIN {X 0,Y 368.933,Z 470.527,A -85,B 0,C 180,E1 -12891.219,E2 -12891.219} C_VEL
LIN {X 0,Y 368.962,Z 470.524,A -85,B 0,C 180,E1 -12894.775,E2 -12894.775} C_VEL
LIN {X 0,Y 368.967,Z 470.523,A -85,B 0,C 180,E1 -12897.203,E2 -12897.203} C_VEL
LIN {X 0,Y 368.932,Z 470.527,A -85,B 0,C 180,E1 -12900.953,E2 -12900.953} C_VEL
LIN {X 0,Y 368.932,Z 470.527,A -85,B 0,C 180,E1 -12905.001,E2 -12905.001} C_VEL
LIN {X 0,Y 368.913,Z 470.53,A -85,B 0,C 180,E1 -12908.64,E2 -12908.64} C_VEL
LIN {X 0,Y 368.882,Z 470.532,A -85,B 0,C 180,E1 -12910.768,E2 -12910.768} C_VEL
LIN {X 0,Y 368.177,Z 470.625,A -85,B 0,C 180,E1 -12911.679,E2 -12911.679} C_VEL
LIN {X 0,Y 365.283,Z 470.982,A -85,B 0,C 180,E1 -12913.161,E2 -12913.161} C_VEL
LIN {X 0,Y 362.877,Z 471.282,A -85,B 0,C 180,E1 -12914.359,E2 -12914.359} C_VEL
LIN {X 0,Y 361.882,Z 471.407,A -85,B 0,C 180,E1 -12915.286,E2 -12915.286} C_VEL
LIN {X 0,Y 361.819,Z 471.417,A -85,B 0,C 180,E1 -12915.6,E2 -12915.6} C_VEL
LIN {X 0,Y 361.838,Z 471.412,A -85,B 0,C 180,E1 -12919.244,E2 -12919.244} C_VEL
LIN {X 0,Y 361.866,Z 471.407,A -85,B 0,C 180,E1 -12922.776,E2 -12922.776} C_VEL
LIN {X 0,Y 361.857,Z 471.413,A -85,B 0,C 180,E1 -12925.719,E2 -12925.719} C_VEL
LIN {X 0,Y 361.876,Z 471.41,A -85,B 0,C 180,E1 -12929.672,E2 -12929.672} C_VEL
LIN {X 0,Y 361.956,Z 471.4,A -85,B 0,C 180,E1 -12933.475,E2 -12933.475} C_VEL
LIN {X 0,Y 361.892,Z 471.406,A -85,B 0,C 180,E1 -12937.144,E2 -12937.144} C_VEL
LIN {X 0,Y 361.922,Z 471.4,A -85,B 0,C 180,E1 -12940.724,E2 -12940.724} C_VEL
LIN {X 0,Y 361.947,Z 471.398,A -85,B 0,C 180,E1 -12944.226,E2 -12944.226} C_VEL
LIN {X 0,Y 362,Z 471.39,A -85,B 0,C 180,E1 -12946.527,E2 -12946.527} C_VEL
LIN {X 0,Y 362.032,Z 471.389,A -85,B 0,C 180,E1 -12949.938,E2 -12949.938} C_VEL
LIN {X 0,Y 362.152,Z 471.372,A -85,B 0,C 180,E1 -12952.192,E2 -12952.192} C_VEL
LIN {X 0,Y 362.119,Z 471.375,A -85,B 0,C 180,E1 -12954.431,E2 -12954.431} C_VEL
LIN {X 0,Y 362.283,Z 471.359,A -85,B 0,C 180,E1 -12957.776,E2 -12957.776} C_VEL
LIN {X 0,Y 362.429,Z 471.339,A -85,B 0,C 180,E1 -12960,E2 -12960} C_VEL
LIN {X 0,Y 362.281,Z 471.355,A -85,B 0,C 180,E1 -12962.223,E2 -12962.223} C_VEL
LIN {X 0,Y 362.173,Z 471.369,A -85,B 0,C 180,E1 -12966.686,E2 -12966.686} C_VEL
LIN {X 0,Y 362.074,Z 471.383,A -85,B 0,C 180,E1 -12968.933,E2 -12968.933} C_VEL
LIN {X 0,Y 361.96,Z 471.395,A -85,B 0,C 180,E1 -12972.332,E2 -12972.332} C_VEL
LIN {X 0,Y 361.962,Z 471.395,A -85,B 0,C 180,E1 -12974.62,E2 -12974.62} C_VEL
LIN {X 0,Y 361.956,Z 471.396,A -85,B 0,C 180,E1 -12978.099,E2 -12978.099} C_VEL
LIN {X 0,Y 361.892,Z 471.407,A -85,B 0,C 180,E1 -12981.653,E2 -12981.653} C_VEL
LIN {X 0,Y 361.928,Z 471.404,A -85,B 0,C 180,E1 -12985.29,E2 -12985.29} C_VEL
LIN {X 0,Y 361.908,Z 471.404,A -85,B 0,C 180,E1 -12987.779,E2 -12987.779} C_VEL
LIN {X 0,Y 361.838,Z 471.413,A -85,B 0,C 180,E1 -12991.629,E2 -12991.629} C_VEL
LIN {X 0,Y 361.874,Z 471.41,A -85,B 0,C 180,E1 -12995.345,E2 -12995.345} C_VEL
LIN {X 0,Y 361.873,Z 471.409,A -85,B 0,C 180,E1 -12999.027,E2 -12999.027} C_VEL
LIN {X 0,Y 361.883,Z 471.405,A -85,B 0,C 180,E1 -13002.44,E2 -13002.44} C_VEL
LIN {X 0,Y 361.907,Z 471.465,A -85,B 0,C 180,E1 -13005.646,E2 -13005.646} C_VEL
LIN {X 0,Y 362.906,Z 477.144,A -85,B 0,C 180,E1 -13009.049,E2 -13009.049} C_VEL
LIN {X 0,Y 363.908,Z 482.933,A -85,B 0,C 180,E1 -13012.356,E2 -13012.356} C_VEL
LIN {X 0,Y 364.099,Z 486.256,A -85,B 0,C 180,E1 -13014.165,E2 -13014.165} C_VEL
LIN {X 0,Y 363.593,Z 491.147,A -85,B 0,C 180,E1 -13016.707,E2 -13016.707} C_VEL
LIN {X 0,Y 362.747,Z 498.977,A -85,B 0,C 180,E1 -13020.674,E2 -13020.674} C_VEL
LIN {X 0,Y 362.042,Z 505.913,A -85,B 0,C 180,E1 -13024.102,E2 -13024.102} C_VEL
LIN {X 0,Y 361.434,Z 513.346,A -85,B 0,C 180,E1 -13027.718,E2 -13027.718} C_VEL
LIN {X 0,Y 361.053,Z 520.128,A -85,B 0,C 180,E1 -13030.972,E2 -13030.972} C_VEL
LIN {X 0,Y 362.731,Z 533.604,A -85,B 0,C 180,E1 -13031.595,E2 -13031.595} C_VEL
LIN {X 0,Y 364.32,Z 547.213,A -85,B 0,C 180,E1 -13032.457,E2 -13032.457} C_VEL
LIN {X 0,Y 364.953,Z 556.847,A -85,B 0,C 180,E1 -13033.211,E2 -13033.211} C_VEL
LIN {X 0,Y 364.017,Z 568.776,A -85,B 0,C 180,E1 -13034.318,E2 -13034.318} C_VEL
LIN {X 0,Y 363.086,Z 579.547,A -85,B 0,C 180,E1 -13035.569,E2 -13035.569} C_VEL
LIN {X 0,Y 362.359,Z 588.408,A -85,B 0,C 180,E1 -13036.827,E2 -13036.827} C_VEL
LIN {X 0,Y 361.725,Z 596.612,A -85,B 0,C 180,E1 -13038.229,E2 -13038.229} C_VEL
LIN {X 0,Y 361.115,Z 604.683,A -85,B 0,C 180,E1 -13039.912,E2 -13039.912} C_VEL
LIN {X 0,Y 360.76,Z 611.174,A -85,B 0,C 180,E1 -13041.599,E2 -13041.599} C_VEL
LIN {X 0,Y 360.568,Z 616.296,A -85,B 0,C 180,E1 -13043.284,E2 -13043.284} C_VEL
LIN {X 0,Y 360.545,Z 620.233,A -85,B 0,C 180,E1 -13044.968,E2 -13044.968} C_VEL
LIN {X 0,Y 360.426,Z 623.065,A -85,B 0,C 180,E1 -13046.647,E2 -13046.647} C_VEL
LIN {X 0,Y 360.559,Z 624.382,A -85,B 0,C 180,E1 -13047.766,E2 -13047.766} C_VEL
LIN {X 0,Y 360.539,Z 625.268,A -85,B 0,C 180,E1 -13048.883,E2 -13048.883} C_VEL
LIN {X 0,Y 360.528,Z 625.737,A -85,B 0,C 180,E1 -13050,E2 -13050} C_VEL
LIN {X 0,Y 360.53,Z 625.743,A -85,B 0,C 180,E1 -13051.117,E2 -13051.117} C_VEL
LIN {X 0,Y 360.47,Z 625.321,A -85,B 0,C 180,E1 -13052.235,E2 -13052.235} C_VEL
LIN {X 0,Y 360.379,Z 624.492,A -85,B 0,C 180,E1 -13053.354,E2 -13053.354} C_VEL
LIN {X 0,Y 360.414,Z 623.25,A -85,B 0,C 180,E1 -13054.474,E2 -13054.474} C_VEL
LIN {X 0,Y 360.388,Z 620.857,A -85,B 0,C 180,E1 -13055.978,E2 -13055.978} C_VEL
LIN {X 0,Y 360.658,Z 616.812,A -85,B 0,C 180,E1 -13057.84,E2 -13057.84} C_VEL
LIN {X 0,Y 361.013,Z 612,A -85,B 0,C 180,E1 -13059.525,E2 -13059.525} C_VEL
LIN {X 0,Y 361.732,Z 604.839,A -85,B 0,C 180,E1 -13061.487,E2 -13061.487} C_VEL
LIN {X 0,Y 362.702,Z 597.211,A -85,B 0,C 180,E1 -13063.161,E2 -13063.161} C_VEL
LIN {X 0,Y 363.778,Z 588.056,A -85,B 0,C 180,E1 -13064.814,E2 -13064.814} C_VEL
LIN {X 0,Y 365.315,Z 577.519,A -85,B 0,C 180,E1 -13066.342,E2 -13066.342} C_VEL
LIN {X 0,Y 366.942,Z 566.051,A -85,B 0,C 180,E1 -13067.701,E2 -13067.701} C_VEL
LIN {X 0,Y 367.778,Z 557.855,A -85,B 0,C 180,E1 -13068.524,E2 -13068.524} C_VEL
LIN {X 0,Y 367.562,Z 544.694,A -85,B 0,C 180,E1 -13069.745,E2 -13069.745} C_VEL
LIN {X 0,Y 366.194,Z 533.926,A -85,B 0,C 180,E1 -13070.663,E2 -13070.663} C_VEL
LIN {X 0,Y 363.437,Z 521.59,A -85,B 0,C 180,E1 -13071.683,E2 -13071.683} C_VEL
LIN {X 0,Y 361.53,Z 514.575,A -85,B 0,C 180,E1 -13072.258,E2 -13072.258} C_VEL
LIN {X 0,Y 362.195,Z 507.604,A -85,B 0,C 180,E1 -13075.887,E2 -13075.887} C_VEL
LIN {X 0,Y 362.988,Z 501.38,A -85,B 0,C 180,E1 -13079.393,E2 -13079.393} C_VEL
LIN {X 0,Y 363.881,Z 496.022,A -85,B 0,C 180,E1 -13082.738,E2 -13082.738} C_VEL
LIN {X 0,Y 364.561,Z 492.337,A -85,B 0,C 180,E1 -13085.334,E2 -13085.334} C_VEL
LIN {X 0,Y 364.845,Z 489.292,A -85,B 0,C 180,E1 -13087.835,E2 -13087.835} C_VEL
LIN {X 0,Y 364.662,Z 487.532,A -85,B 0,C 180,E1 -13089.565,E2 -13089.565} C_VEL
LIN {X 0,Y 364.243,Z 484.838,A -85,B 0,C 180,E1 -13092.844,E2 -13092.844} C_VEL
LIN {X 0,Y 363.952,Z 483.02,A -85,B 0,C 180,E1 -13095.959,E2 -13095.959} C_VEL
LIN {X 0,Y 363.68,Z 481.94,A -85,B 0,C 180,E1 -13098.926,E2 -13098.926} C_VEL
LIN {X 0,Y 363.457,Z 481.393,A -85,B 0,C 180,E1 -13102.448,E2 -13102.448} C_VEL
LIN {X 0,Y 363.297,Z 481.431,A -85,B 0,C 180,E1 -13104.525,E2 -13104.525} C_VEL
LIN {X 0,Y 362.988,Z 481.817,A -85,B 0,C 180,E1 -13107.172,E2 -13107.172} C_VEL
LIN {X 0,Y 362.66,Z 482.509,A -85,B 0,C 180,E1 -13109.745,E2 -13109.745} C_VEL
LIN {X 0,Y 362.172,Z 483.969,A -85,B 0,C 180,E1 -13113.492,E2 -13113.492} C_VEL
LIN {X 0,Y 361.827,Z 485.789,A -85,B 0,C 180,E1 -13117.141,E2 -13117.141} C_VEL
LIN {X 0,Y 361.789,Z 486.293,A -85,B 0,C 180,E1 -13117.957,E2 -13117.957} C_VEL
LIN {X 0,Y 362.879,Z 489.186,A -85,B 0,C 180,E1 -13118.245,E2 -13118.245} C_VEL
LIN {X 0,Y 367.04,Z 498.795,A -85,B 0,C 180,E1 -13119.298,E2 -13119.298} C_VEL
LIN {X 0,Y 370.395,Z 510.16,A -85,B 0,C 180,E1 -13120.511,E2 -13120.511} C_VEL
LIN {X 0,Y 370.852,Z 511.933,A -85,B 0,C 180,E1 -13120.704,E2 -13120.704} C_VEL
LIN {X 0,Y 369.859,Z 522.348,A -85,B 0,C 180,E1 -13121.628,E2 -13121.628} C_VEL
LIN {X 0,Y 368.292,Z 534.154,A -85,B 0,C 180,E1 -13122.903,E2 -13122.903} C_VEL
LIN {X 0,Y 366.908,Z 543.703,A -85,B 0,C 180,E1 -13124.16,E2 -13124.16} C_VEL
LIN {X 0,Y 365.343,Z 553.765,A -85,B 0,C 180,E1 -13125.803,E2 -13125.803} C_VEL
LIN {X 0,Y 364.124,Z 561.913,A -85,B 0,C 180,E1 -13127.459,E2 -13127.459} C_VEL
LIN {X 0,Y 363.027,Z 569.43,A -85,B 0,C 180,E1 -13129.402,E2 -13129.402} C_VEL
LIN {X 0,Y 362.217,Z 574.551,A -85,B 0,C 180,E1 -13131.071,E2 -13131.071} C_VEL
LIN {X 0,Y 361.516,Z 578.789,A -85,B 0,C 180,E1 -13132.863,E2 -13132.863} C_VEL
LIN {X 0,Y 361.14,Z 581.463,A -85,B 0,C 180,E1 -13134.416,E2 -13134.416} C_VEL
LIN {X 0,Y 361.073,Z 582.881,A -85,B 0,C 180,E1 -13135.535,E2 -13135.535} C_VEL
LIN {X 0,Y 360.865,Z 583.877,A -85,B 0,C 180,E1 -13136.651,E2 -13136.651} C_VEL
LIN {X 0,Y 360.707,Z 584.46,A -85,B 0,C 180,E1 -13137.767,E2 -13137.767} C_VEL
LIN {X 0,Y 360.59,Z 584.65,A -85,B 0,C 180,E1 -13138.883,E2 -13138.883} C_VEL
LIN {X 0,Y 360.531,Z 584.441,A -85,B 0,C 180,E1 -13140,E2 -13140} C_VEL
LIN {X 0,Y 360.549,Z 583.78,A -85,B 0,C 180,E1 -13141.117,E2 -13141.117} C_VEL
LIN {X 0,Y 360.612,Z 582.71,A -85,B 0,C 180,E1 -13142.234,E2 -13142.234} C_VEL
LIN {X 0,Y 360.608,Z 581.24,A -85,B 0,C 180,E1 -13143.352,E2 -13143.352} C_VEL
LIN {X 0,Y 360.752,Z 578.186,A -85,B 0,C 180,E1 -13145.03,E2 -13145.03} C_VEL
LIN {X 0,Y 361.041,Z 573.56,A -85,B 0,C 180,E1 -13146.894,E2 -13146.894} C_VEL
LIN {X 0,Y 361.371,Z 567.776,A -85,B 0,C 180,E1 -13148.669,E2 -13148.669} C_VEL
LIN {X 0,Y 361.898,Z 560.915,A -85,B 0,C 180,E1 -13150.349,E2 -13150.349} C_VEL
LIN {X 0,Y 362.575,Z 552.453,A -85,B 0,C 180,E1 -13152.027,E2 -13152.027} C_VEL
LIN {X 0,Y 363.328,Z 543.811,A -85,B 0,C 180,E1 -13153.422,E2 -13153.422} C_VEL
LIN {X 0,Y 364.317,Z 532.254,A -85,B 0,C 180,E1 -13154.937,E2 -13154.937} C_VEL
LIN {X 0,Y 365.003,Z 521.564,A -85,B 0,C 180,E1 -13156.069,E2 -13156.069} C_VEL
LIN {X 0,Y 365.965,Z 508.296,A -85,B 0,C 180,E1 -13157.171,E2 -13157.171} C_VEL
LIN {X 0,Y 365.797,Z 504.253,A -85,B 0,C 180,E1 -13157.465,E2 -13157.465} C_VEL
LIN {X 0,Y 363.253,Z 492.197,A -85,B 0,C 180,E1 -13158.287,E2 -13158.287} C_VEL
LIN {X 0,Y 360.725,Z 480.007,A -85,B 0,C 180,E1 -13158.936,E2 -13158.936} C_VEL
LIN {X 0,Y 360.763,Z 476.05,A -85,B 0,C 180,E1 -13162.931,E2 -13162.931} C_VEL
LIN {X 0,Y 360.903,Z 472.501,A -85,B 0,C 180,E1 -13166.609,E2 -13166.609} C_VEL
LIN {X 0,Y 360.94,Z 471.529,A -85,B 0,C 180,E1 -13167.86,E2 -13167.86} C_VEL
LIN {X 0,Y 361.298,Z 471.478,A -85,B 0,C 180,E1 -13171.141,E2 -13171.141} C_VEL
LIN {X 0,Y 361.635,Z 471.441,A -85,B 0,C 180,E1 -13174.305,E2 -13174.305} C_VEL
LIN {X 0,Y 361.838,Z 471.41,A -85,B 0,C 180,E1 -13177.217,E2 -13177.217} C_VEL
LIN {X 0,Y 361.859,Z 471.41,A -85,B 0,C 180,E1 -13179.861,E2 -13179.861} C_VEL
LIN {X 0,Y 361.84,Z 471.412,A -85,B 0,C 180,E1 -13182.829,E2 -13182.829} C_VEL
LIN {X 0,Y 361.823,Z 471.415,A -85,B 0,C 180,E1 -13185.947,E2 -13185.947} C_VEL
LIN {X 0,Y 361.84,Z 471.41,A -85,B 0,C 180,E1 -13189.245,E2 -13189.245} C_VEL
LIN {X 0,Y 361.869,Z 471.407,A -85,B 0,C 180,E1 -13192.777,E2 -13192.777} C_VEL
LIN {X 0,Y 361.86,Z 471.41,A -85,B 0,C 180,E1 -13195.72,E2 -13195.72} C_VEL
LIN {X 0,Y 361.878,Z 471.407,A -85,B 0,C 180,E1 -13199.672,E2 -13199.672} C_VEL
LIN {X 0,Y 361.959,Z 471.396,A -85,B 0,C 180,E1 -13203.475,E2 -13203.475} C_VEL
LIN {X 0,Y 361.896,Z 471.403,A -85,B 0,C 180,E1 -13207.145,E2 -13207.145} C_VEL
LIN {X 0,Y 361.926,Z 471.401,A -85,B 0,C 180,E1 -13210.724,E2 -13210.724} C_VEL
LIN {X 0,Y 361.951,Z 471.401,A -85,B 0,C 180,E1 -13214.226,E2 -13214.226} C_VEL
LIN {X 0,Y 362.004,Z 471.392,A -85,B 0,C 180,E1 -13216.528,E2 -13216.528} C_VEL
LIN {X 0,Y 362.035,Z 471.39,A -85,B 0,C 180,E1 -13219.938,E2 -13219.938} C_VEL
LIN {X 0,Y 362.162,Z 471.37,A -85,B 0,C 180,E1 -13223.313,E2 -13223.313} C_VEL
LIN {X 0,Y 362.286,Z 471.358,A -85,B 0,C 180,E1 -13227.776,E2 -13227.776} C_VEL
LIN {X 0,Y 362.432,Z 471.342,A -85,B 0,C 180,E1 -13230,E2 -13230} C_VEL
LIN {X 0,Y 362.286,Z 471.359,A -85,B 0,C 180,E1 -13232.223,E2 -13232.223} C_VEL
LIN {X 0,Y 362.145,Z 471.372,A -85,B 0,C 180,E1 -13236.686,E2 -13236.686} C_VEL
LIN {X 0,Y 362.036,Z 471.39,A -85,B 0,C 180,E1 -13240.062,E2 -13240.062} C_VEL
LIN {X 0,Y 362.002,Z 471.395,A -85,B 0,C 180,E1 -13243.899,E2 -13243.899} C_VEL
LIN {X 0,Y 361.972,Z 471.398,A -85,B 0,C 180,E1 -13247.938,E2 -13247.938} C_VEL
